C09099=1090.763,165.614,-68.521,176.010,19.399,152.921
C09100=1090.757,165.365,-68.500,176.007,19.398,152.921
C09101=1090.752,165.116,-68.478,176.005,19.397,152.921
C09102=1090.746,164.867,-68.456,176.002,19.396,152.921
C09103=1090.741,164.618,-68.434,175.999,19.395,152.922
C09104=1090.735,164.369,-68.413,175.996,19.394,152.922
C09105=1090.731,164.119,-68.391,175.994,19.392,152.922
C09106=1090.725,163.871,-68.370,175.991,19.391,152.922
C09107=1090.719,163.622,-68.348,175.988,19.390,152.923
C09108=1090.714,163.373,-68.327,175.986,19.389,152.923
C09109=1090.709,163.124,-68.305,175.983,19.388,152.923
C09110=1090.703,162.874,-68.284,175.981,19.387,152.923
C09111=1090.698,162.626,-68.263,175.978,19.386,152.923
C09112=1090.692,162.377,-68.241,175.976,19.385,152.924
C09113=1090.687,162.128,-68.219,175.973,19.383,152.924
C09114=1090.681,161.879,-68.198,175.970,19.382,152.924
C09115=1090.676,161.629,-68.176,175.967,19.381,152.924
C09116=1090.671,161.381,-68.155,175.965,19.380,152.925
C09117=1090.665,161.132,-68.134,175.962,19.379,152.925
C09118=1090.659,160.882,-68.113,175.959,19.378,152.925
C09119=1090.654,160.634,-68.092,175.957,19.377,152.925
C09120=1090.647,160.385,-68.070,175.955,19.376,152.926
C09121=1090.642,160.108,-68.046,175.952,19.375,152.926
C09122=1090.635,159.831,-68.023,175.948,19.373,152.926
C09123=1090.629,159.553,-67.999,175.946,19.372,152.926
C09124=1090.623,159.277,-67.975,175.943,19.371,152.927
C09125=1090.617,159.028,-67.954,175.940,19.370,152.927
C09126=1090.612,158.778,-67.933,175.937,19.369,152.927
C09127=1090.606,158.530,-67.912,175.935,19.368,152.927
C09128=1090.600,158.280,-67.891,175.932,19.367,152.927
C09129=1090.595,158.031,-67.870,175.930,19.366,152.928
C09130=1090.590,157.783,-67.848,175.927,19.365,152.928
C09131=1090.584,157.533,-67.827,175.925,19.364,152.928
C09132=1090.578,157.284,-67.806,175.922,19.362,152.928
C09133=1090.573,157.035,-67.785,175.919,19.361,152.929
C09134=1090.567,156.786,-67.763,175.916,19.360,152.929
C09135=1090.562,156.537,-67.743,175.914,19.359,152.929
C09136=1090.556,156.288,-67.722,175.912,19.358,152.929
C09137=1090.550,156.039,-67.700,175.909,19.357,152.929
C09138=1090.545,155.790,-67.679,175.906,19.356,152.930
C09139=1090.539,155.541,-67.658,175.904,19.355,152.930
C09140=1090.533,155.292,-67.637,175.901,19.353,152.930
C09141=1090.528,155.043,-67.616,175.898,19.352,152.930
C09142=1090.522,154.794,-67.595,175.896,19.351,152.931
C09143=1090.517,154.544,-67.574,175.894,19.351,152.931
C09144=1090.511,154.296,-67.553,175.891,19.349,152.931
C09145=1090.506,154.047,-67.533,175.888,19.348,152.931
C09146=1090.500,153.797,-67.511,175.886,19.347,152.932
C09147=1090.494,153.548,-67.490,175.883,19.346,152.932
C09148=1090.489,153.300,-67.469,175.880,19.344,152.932
C09149=1090.483,153.051,-67.449,175.878,19.344,152.932
C09150=1090.478,152.801,-67.428,175.876,19.343,152.932
C09151=1090.472,152.552,-67.406,175.873,19.341,152.933
C09152=1090.467,152.303,-67.386,175.870,19.340,152.933
C09153=1090.461,152.053,-67.365,175.868,19.339,152.933
C09154=1090.455,151.805,-67.344,175.865,19.338,152.933
C09155=1090.449,151.556,-67.324,175.863,19.337,152.933
C09156=1090.444,151.307,-67.303,175.860,19.336,152.934
C09157=1090.438,151.058,-67.282,175.858,19.334,152.934
C09158=1090.433,150.809,-67.261,175.855,19.333,152.934
C09159=1090.427,150.559,-67.240,175.852,19.332,152.934
C09160=1090.422,150.311,-67.219,175.850,19.331,152.934
C09161=1090.416,150.061,-67.198,175.848,19.330,152.935
C09162=1090.411,149.812,-67.178,175.845,19.329,152.935
C09163=1090.404,149.564,-67.157,175.843,19.328,152.935
C09164=1090.399,149.315,-67.136,175.840,19.327,152.935
C09165=1090.394,149.066,-67.116,175.837,19.325,152.936
C09166=1090.388,148.816,-67.095,175.835,19.324,152.936
C09167=1090.383,148.567,-67.074,175.833,19.323,152.936
C09168=1090.377,148.318,-67.053,175.830,19.322,152.936
C09169=1090.371,148.069,-67.033,175.827,19.321,152.936
C09170=1090.366,147.820,-67.013,175.825,19.320,152.937
C09171=1090.360,147.570,-66.992,175.822,19.318,152.937
C09172=1090.355,147.321,-66.971,175.820,19.318,152.937
C09173=1090.349,147.073,-66.951,175.817,19.317,152.937
C09174=1090.343,146.824,-66.930,175.815,19.315,152.937
C09175=1090.338,146.574,-66.909,175.812,19.314,152.938
C09176=1090.332,146.325,-66.889,175.809,19.312,152.938
C09177=1090.326,146.076,-66.869,175.808,19.312,152.938
C09178=1090.321,145.827,-66.848,175.805,19.311,152.938
C09179=1090.316,145.578,-66.827,175.802,19.309,152.938
C09180=1090.310,145.329,-66.807,175.799,19.308,152.939
C09181=1090.304,145.079,-66.787,175.797,19.307,152.939
C09182=1090.298,144.831,-66.765,175.795,19.306,152.939
C09183=1090.292,144.582,-66.745,175.792,19.305,152.939
C09184=1090.287,144.333,-66.725,175.790,19.303,152.939
C09185=1090.280,144.055,-66.702,175.787,19.302,152.940
C09186=1090.275,143.778,-66.679,175.784,19.301,152.940
C09187=1090.268,143.501,-66.657,175.782,19.300,152.940
C09188=1090.262,143.223,-66.634,175.779,19.298,152.940
C09189=1090.256,142.974,-66.614,175.776,19.297,152.940
C09190=1090.251,142.725,-66.594,175.774,19.296,152.940
C09191=1090.246,142.476,-66.573,175.771,19.295,152.941
C09192=1090.240,142.227,-66.553,175.769,19.293,152.941
C09193=1090.235,141.978,-66.533,175.767,19.292,152.941
C09194=1090.229,141.729,-66.512,175.764,19.291,152.941
C09195=1090.223,141.480,-66.492,175.761,19.290,152.941
C09196=1090.217,141.230,-66.471,175.759,19.288,152.942
C09197=1090.212,140.981,-66.451,175.757,19.288,152.942
C09198=1090.206,140.732,-66.431,175.754,19.286,152.942
C09199=1090.201,140.483,-66.410,175.752,19.285,152.942
C09200=1090.195,140.234,-66.390,175.749,19.284,152.942
C09201=1090.190,139.985,-66.370,175.746,19.283,152.943
C09202=1090.184,139.736,-66.350,175.745,19.282,152.943
C09203=1090.179,139.487,-66.330,175.742,19.280,152.943
C09204=1090.173,139.238,-66.310,175.739,19.279,152.943
C09205=1090.168,138.989,-66.289,175.737,19.277,152.943
C09206=1090.162,138.740,-66.269,175.735,19.277,152.943
C09207=1090.156,138.491,-66.249,175.732,19.275,152.944
C09208=1090.151,138.241,-66.230,175.730,19.274,152.944
C09209=1090.145,137.992,-66.209,175.727,19.273,152.944
C09210=1090.139,137.743,-66.189,175.725,19.272,152.944
C09211=1090.133,137.494,-66.168,175.723,19.271,152.944
C09212=1090.127,137.245,-66.148,175.720,19.270,152.945
C09213=1090.123,136.995,-66.128,175.717,19.268,152.945
C09214=1090.117,136.746,-66.108,175.715,19.266,152.945
C09215=1090.111,136.497,-66.088,175.713,19.266,152.945
C09216=1090.105,136.248,-66.068,175.710,19.264,152.945
C09217=1090.100,135.999,-66.049,175.708,19.263,152.945
C09218=1090.094,135.750,-66.028,175.705,19.262,152.946
C09219=1090.088,135.501,-66.008,175.703,19.261,152.946
C09220=1090.083,135.251,-65.988,175.701,19.260,152.946
C09221=1090.077,135.002,-65.968,175.698,19.258,152.946
C09222=1090.071,134.753,-65.948,175.695,19.257,152.946
C09223=1090.066,134.504,-65.928,175.694,19.256,152.946
C09224=1090.060,134.255,-65.909,175.691,19.254,152.946
C09225=1090.054,134.006,-65.889,175.688,19.253,152.947
C09226=1090.050,133.756,-65.869,175.686,19.252,152.947
C09227=1090.044,133.508,-65.849,175.684,19.251,152.947
C09228=1090.038,133.258,-65.828,175.681,19.250,152.947
C09229=1090.033,133.009,-65.809,175.679,19.248,152.947
C09230=1090.027,132.760,-65.789,175.676,19.247,152.947
C09231=1090.022,132.510,-65.769,175.674,19.246,152.948
C09232=1090.016,132.262,-65.749,175.672,19.245,152.948
C09233=1090.010,132.012,-65.730,175.669,19.243,152.948
C09234=1090.005,131.763,-65.709,175.667,19.242,152.948
C09235=1089.999,131.514,-65.689,175.665,19.241,152.948
C09236=1089.993,131.265,-65.670,175.662,19.239,152.948
C09237=1089.987,131.016,-65.650,175.660,19.238,152.949
C09238=1089.981,130.767,-65.631,175.658,19.237,152.949
C09239=1089.975,130.518,-65.611,175.655,19.236,152.949
C09240=1089.970,130.268,-65.591,175.653,19.235,152.949
C09241=1089.965,130.020,-65.572,175.650,19.233,152.949
C09242=1089.959,129.770,-65.552,175.648,19.233,152.950
C09243=1089.953,129.522,-65.532,175.646,19.231,152.950
C09244=1089.948,129.272,-65.513,175.643,19.229,152.950
C09245=1089.942,129.023,-65.493,175.641,19.229,152.950
C09246=1089.936,128.774,-65.474,175.639,19.227,152.950
C09247=1089.931,128.524,-65.454,175.636,19.226,152.950
C09248=1089.925,128.275,-65.434,175.634,19.224,152.950
C09249=1089.919,127.998,-65.413,175.631,19.223,152.951
C09250=1089.911,127.720,-65.391,175.628,19.222,152.951
C09251=1089.906,127.443,-65.369,175.626,19.220,152.951
C09252=1089.899,127.166,-65.347,175.623,19.219,152.951
C09253=1089.894,126.917,-65.328,175.621,19.218,152.951
C09254=1089.888,126.668,-65.308,175.619,19.217,152.951
C09255=1089.883,126.418,-65.288,175.616,19.215,152.952
C09256=1089.878,126.169,-65.269,175.613,19.214,152.952
C09257=1089.872,125.920,-65.249,175.612,19.213,152.952
C09258=1089.866,125.671,-65.230,175.609,19.211,152.952
C09259=1089.860,125.422,-65.211,175.607,19.210,152.952
C09260=1089.854,125.173,-65.191,175.605,19.209,152.952
C09261=1089.848,124.923,-65.172,175.602,19.208,152.952
C09262=1089.843,124.674,-65.152,175.600,19.206,152.953
C09263=1089.837,124.424,-65.133,175.598,19.205,152.953
C09264=1089.832,124.176,-65.114,175.596,19.204,152.953
C09265=1089.826,123.927,-65.094,175.593,19.202,152.953
C09266=1089.820,123.677,-65.075,175.590,19.201,152.953
C09267=1089.815,123.428,-65.056,175.589,19.200,152.953
C09268=1089.809,123.179,-65.036,175.586,19.198,152.953
C09269=1089.804,122.929,-65.016,175.584,19.197,152.954
C09270=1089.799,122.681,-64.997,175.582,19.196,152.954
C09271=1089.793,122.431,-64.978,175.579,19.194,152.954
C09272=1089.787,122.182,-64.959,175.577,19.193,152.954
C09273=1089.781,121.933,-64.939,175.575,19.192,152.954
C09274=1089.776,121.684,-64.919,175.572,19.191,152.954
C09275=1089.770,121.435,-64.901,175.570,19.189,152.954
C09276=1089.765,121.185,-64.881,175.567,19.188,152.954
C09277=1089.759,120.936,-64.862,175.566,19.186,152.955
C09278=1089.753,120.687,-64.843,175.563,19.185,152.955
C09279=1089.748,120.438,-64.824,175.561,19.183,152.955
C09280=1089.742,120.189,-64.804,175.559,19.182,152.955
C09281=1089.737,119.940,-64.785,175.556,19.181,152.955
C09282=1089.731,119.690,-64.766,175.554,19.179,152.955
C09283=1089.726,119.441,-64.747,175.552,19.178,152.955
C09284=1089.720,119.192,-64.727,175.550,19.177,152.955
C09285=1089.715,118.943,-64.708,175.547,19.176,152.956
C09286=1089.709,118.693,-64.689,175.545,19.175,152.956
C09287=1089.704,118.444,-64.670,175.543,19.173,152.956
C09288=1089.698,118.195,-64.651,175.540,19.171,152.956
C09289=1089.692,117.946,-64.632,175.538,19.170,152.956
C09290=1089.687,117.696,-64.612,175.536,19.169,152.956
C09291=1089.682,117.447,-64.593,175.533,19.167,152.956
C09292=1089.676,117.198,-64.574,175.532,19.166,152.956
C09293=1089.669,116.949,-64.556,175.529,19.165,152.957
C09294=1089.664,116.700,-64.537,175.527,19.163,152.957
C09295=1089.659,116.451,-64.517,175.525,19.162,152.957
C09296=1089.653,116.201,-64.498,175.523,19.160,152.957
C09297=1089.648,115.953,-64.479,175.520,19.159,152.957
C09298=1089.642,115.703,-64.460,175.518,19.158,152.957
C09299=1089.637,115.454,-64.441,175.516,19.156,152.957
C09300=1089.631,115.205,-64.422,175.513,19.154,152.957
C09301=1089.626,114.956,-64.403,175.512,19.153,152.957
C09302=1089.620,114.706,-64.383,175.509,19.152,152.957
C09303=1089.615,114.457,-64.365,175.507,19.150,152.958
C09304=1089.610,114.207,-64.346,175.505,19.149,152.958
C09305=1089.603,113.958,-64.327,175.503,19.148,152.958
C09306=1089.598,113.709,-64.308,175.500,19.146,152.958
C09307=1089.592,113.460,-64.289,175.498,19.145,152.958
C09308=1089.587,113.211,-64.270,175.496,19.144,152.958
C09309=1089.581,112.962,-64.252,175.493,19.142,152.958
C09310=1089.575,112.713,-64.232,175.492,19.141,152.958
C09311=1089.570,112.463,-64.214,175.489,19.139,152.958
C09312=1089.565,112.214,-64.195,175.487,19.138,152.959
C09313=1089.558,111.937,-64.174,175.484,19.136,152.959
C09314=1089.551,111.659,-64.153,175.481,19.135,152.959
C09315=1089.545,111.382,-64.132,175.479,19.133,152.959
C09316=1089.539,111.104,-64.112,175.477,19.131,152.959
C09317=1089.534,110.855,-64.093,175.475,19.130,152.959
C09318=1089.527,110.606,-64.074,175.472,19.129,152.959
C09319=1089.522,110.357,-64.055,175.471,19.128,152.959
C09320=1089.517,110.107,-64.037,175.468,19.126,152.959
C09321=1089.511,109.858,-64.018,175.466,19.125,152.960
C09322=1089.505,109.609,-63.999,175.464,19.123,152.960
C09323=1089.499,109.360,-63.981,175.462,19.122,152.960
C09324=1089.494,109.110,-63.962,175.459,19.120,152.960
C09325=1089.488,108.861,-63.943,175.457,19.119,152.960
C09326=1089.482,108.612,-63.925,175.455,19.118,152.960
C09327=1089.477,108.362,-63.906,175.452,19.116,152.960
C09328=1089.471,108.114,-63.888,175.451,19.115,152.960
C09329=1089.465,107.865,-63.869,175.448,19.114,152.960
C09330=1089.460,107.614,-63.850,175.447,19.112,152.960
C09331=1089.454,107.366,-63.832,175.444,19.111,152.961
C09332=1089.448,107.117,-63.813,175.442,19.109,152.961
C09333=1089.443,106.868,-63.795,175.440,19.108,152.961
C09334=1089.437,106.618,-63.776,175.437,19.106,152.961
C09335=1089.431,106.368,-63.758,175.435,19.105,152.961
C09336=1089.426,106.120,-63.739,175.433,19.104,152.961
C09337=1089.420,105.870,-63.720,175.431,19.102,152.961
C09338=1089.415,105.621,-63.702,175.429,19.101,152.961
C09339=1089.409,105.372,-63.683,175.427,19.099,152.961
C09340=1089.404,105.123,-63.665,175.424,19.098,152.961
C09341=1089.398,104.873,-63.646,175.422,19.097,152.962
C09342=1089.392,104.624,-63.628,175.420,19.095,152.961
C09343=1089.387,104.375,-63.609,175.418,19.093,152.962
C09344=1089.381,104.125,-63.591,175.416,19.092,152.962
C09345=1089.375,103.876,-63.572,175.413,19.090,152.962
C09346=1089.369,103.627,-63.554,175.412,19.089,152.962
C09347=1089.364,103.378,-63.536,175.410,19.087,152.962
C09348=1089.358,103.128,-63.518,175.407,19.086,152.962
C09349=1089.353,102.879,-63.499,175.405,19.085,152.962
C09350=1089.347,102.630,-63.481,175.403,19.083,152.962
C09351=1089.342,102.381,-63.462,175.401,19.081,152.962
C09352=1089.336,102.131,-63.443,175.399,19.080,152.962
C09353=1089.331,101.882,-63.425,175.396,19.079,152.962
C09354=1089.325,101.633,-63.407,175.395,19.078,152.963
C09355=1089.320,101.383,-63.389,175.392,19.076,152.963
C09356=1089.313,101.134,-63.370,175.390,19.074,152.963
C09357=1089.309,100.885,-63.352,175.388,19.073,152.963
C09358=1089.302,100.636,-63.334,175.386,19.071,152.963
C09359=1089.297,100.387,-63.316,175.384,19.070,152.963
C09360=1089.291,100.137,-63.298,175.382,19.068,152.963
C09361=1089.285,99.888,-63.279,175.379,19.067,152.963
C09362=1089.279,99.639,-63.261,175.377,19.066,152.963
C09363=1089.274,99.390,-63.242,175.375,19.064,152.963
C09364=1089.268,99.140,-63.225,175.374,19.063,152.963
C09365=1089.263,98.891,-63.207,175.371,19.061,152.963
C09366=1089.257,98.641,-63.188,175.368,19.060,152.964
C09367=1089.251,98.393,-63.170,175.367,19.058,152.963
C09368=1089.245,98.143,-63.152,175.365,19.057,152.964
C09369=1089.240,97.893,-63.134,175.363,19.055,152.964
C09370=1089.235,97.645,-63.116,175.360,19.054,152.964
C09371=1089.228,97.395,-63.098,175.358,19.052,152.964
C09372=1089.223,97.146,-63.080,175.356,19.051,152.964
C09373=1089.218,96.896,-63.062,175.354,19.049,152.964
C09374=1089.212,96.648,-63.043,175.352,19.048,152.964
C09375=1089.206,96.398,-63.026,175.350,19.046,152.964
C09376=1089.201,96.149,-63.007,175.347,19.045,152.964
C09377=1089.194,95.871,-62.988,175.346,19.043,152.964
C09378=1089.188,95.595,-62.967,175.343,19.042,152.964
C09379=1089.181,95.317,-62.947,175.341,19.040,152.964
C09380=1089.175,95.039,-62.927,175.339,19.038,152.964
C09381=1089.169,94.790,-62.909,175.336,19.036,152.965
C09382=1089.164,94.541,-62.891,175.335,19.035,152.965
C09383=1089.159,94.292,-62.873,175.332,19.033,152.965
C09384=1089.153,94.042,-62.855,175.330,19.032,152.965
C09385=1089.147,93.793,-62.838,175.328,19.030,152.965
C09386=1089.142,93.544,-62.820,175.326,19.029,152.965
C09387=1089.136,93.294,-62.801,175.324,19.027,152.965
C09388=1089.131,93.045,-62.784,175.322,19.026,152.965
C09389=1089.125,92.795,-62.766,175.320,19.025,152.965
C09390=1089.119,92.547,-62.748,175.318,19.023,152.965
C09391=1089.113,92.298,-62.730,175.316,19.022,152.965
C09392=1089.108,92.048,-62.712,175.314,19.019,152.965
C09393=1089.102,91.799,-62.694,175.311,19.018,152.965
C09394=1089.097,91.550,-62.676,175.310,19.016,152.965
C09395=1089.091,91.300,-62.658,175.307,19.015,152.965
C09396=1089.085,91.051,-62.641,175.306,19.014,152.965
C09397=1089.080,90.802,-62.623,175.303,19.012,152.965
C09398=1089.074,90.552,-62.605,175.302,19.011,152.965
C09399=1089.069,90.303,-62.587,175.299,19.009,152.965
C09400=1089.063,90.054,-62.570,175.297,19.007,152.966
C09401=1089.057,89.804,-62.552,175.295,19.006,152.966
C09402=1089.052,89.555,-62.534,175.293,19.004,152.966
C09403=1089.045,89.305,-62.516,175.291,19.003,152.966
C09404=1089.040,89.056,-62.499,175.289,19.001,152.966
C09405=1089.034,88.807,-62.481,175.287,19.000,152.966
C09406=1089.028,88.557,-62.463,175.285,18.998,152.966
C09407=1089.023,88.308,-62.446,175.282,18.996,152.966
C09408=1089.017,88.059,-62.428,175.281,18.995,152.966
C09409=1089.011,87.810,-62.410,175.279,18.993,152.966
C09410=1089.006,87.561,-62.393,175.277,18.992,152.966
C09411=1089.000,87.312,-62.375,175.275,18.990,152.966
C09412=1088.994,87.062,-62.357,175.273,18.989,152.966
C09413=1088.989,86.812,-62.340,175.271,18.987,152.966
C09414=1088.983,86.563,-62.323,175.269,18.986,152.966
C09415=1088.977,86.313,-62.305,175.266,18.984,152.966
C09416=1088.972,86.064,-62.287,175.264,18.982,152.966
C09417=1088.966,85.815,-62.270,175.262,18.981,152.967
C09418=1088.961,85.566,-62.252,175.260,18.979,152.967
C09419=1088.954,85.316,-62.234,175.259,18.978,152.967
C09420=1088.949,85.067,-62.217,175.256,18.976,152.967
C09421=1088.943,84.818,-62.200,175.255,18.975,152.967
C09422=1088.937,84.569,-62.183,175.252,18.973,152.967
C09423=1088.931,84.319,-62.165,175.251,18.972,152.967
C09424=1088.926,84.070,-62.147,175.248,18.970,152.967
C09425=1088.920,83.821,-62.130,175.247,18.969,152.967
C09426=1088.915,83.572,-62.113,175.244,18.967,152.967
C09427=1088.909,83.322,-62.095,175.242,18.965,152.967
C09428=1088.903,83.073,-62.077,175.240,18.964,152.967
C09429=1088.898,82.824,-62.060,175.238,18.962,152.967
C09430=1088.893,82.574,-62.043,175.236,18.961,152.967
C09431=1088.887,82.324,-62.025,175.234,18.959,152.967
C09432=1088.881,82.075,-62.007,175.233,18.957,152.967
C09433=1088.876,81.826,-61.990,175.230,18.956,152.967
C09434=1088.870,81.577,-61.973,175.229,18.954,152.967
C09435=1088.864,81.328,-61.956,175.226,18.953,152.967
C09436=1088.858,81.078,-61.938,175.225,18.951,152.967
C09437=1088.853,80.828,-61.921,175.223,18.949,152.967
C09438=1088.847,80.579,-61.904,175.221,18.948,152.967
C09439=1088.842,80.330,-61.886,175.219,18.946,152.967
C09440=1088.837,80.081,-61.869,175.216,18.944,152.967
C09441=1088.830,79.804,-61.850,175.215,18.943,152.967
C09442=1088.824,79.526,-61.830,175.212,18.941,152.967
C09443=1088.817,79.248,-61.811,175.210,18.939,152.967
C09444=1088.811,78.972,-61.792,175.208,18.937,152.967
C09445=1088.805,78.723,-61.775,175.206,18.936,152.967
C09446=1088.800,78.473,-61.758,175.204,18.934,152.967
C09447=1088.795,78.224,-61.740,175.202,18.933,152.967
C09448=1088.788,77.974,-61.724,175.200,18.931,152.967
C09449=1088.783,77.725,-61.706,175.198,18.929,152.967
C09450=1088.777,77.476,-61.689,175.196,18.927,152.967
C09451=1088.772,77.226,-61.672,175.195,18.926,152.967
C09452=1088.766,76.977,-61.655,175.192,18.924,152.968
C09453=1088.760,76.727,-61.637,175.191,18.923,152.968
C09454=1088.754,76.478,-61.620,175.188,18.921,152.968
C09455=1088.748,76.229,-61.604,175.187,18.920,152.968
C09456=1088.743,75.980,-61.586,175.184,18.918,152.968
C09457=1088.738,75.730,-61.569,175.182,18.916,152.968
C09458=1088.731,75.481,-61.552,175.180,18.915,152.968
C09459=1088.726,75.232,-61.535,175.178,18.913,152.968
C09460=1088.720,74.982,-61.517,175.177,18.911,152.968
C09461=1088.714,74.732,-61.501,175.174,18.909,152.968
C09462=1088.708,74.483,-61.484,175.173,18.908,152.968
C09463=1088.703,74.234,-61.467,175.170,18.906,152.968
C09464=1088.697,73.985,-61.450,175.169,18.905,152.968
C09465=1088.692,73.735,-61.433,175.167,18.903,152.968
C09466=1088.686,73.486,-61.415,175.165,18.902,152.968
C09467=1088.680,73.237,-61.399,175.163,18.900,152.968
C09468=1088.675,72.987,-61.382,175.161,18.898,152.968
C09469=1088.669,72.738,-61.364,175.159,18.897,152.968
C09470=1088.663,72.488,-61.348,175.157,18.895,152.968
C09471=1088.658,72.239,-61.331,175.155,18.893,152.968
C09472=1088.652,71.989,-61.314,175.153,18.892,152.968
C09473=1088.646,71.740,-61.297,175.151,18.890,152.968
C09474=1088.641,71.491,-61.280,175.150,18.888,152.968
C09475=1088.635,71.242,-61.264,175.147,18.886,152.968
C09476=1088.630,70.992,-61.247,175.146,18.885,152.968
C09477=1088.624,70.743,-61.229,175.143,18.883,152.968
C09478=1088.618,70.494,-61.213,175.142,18.882,152.968
C09479=1088.613,70.244,-61.196,175.140,18.880,152.968
C09480=1088.607,69.995,-61.179,175.138,18.879,152.968
C09481=1088.602,69.746,-61.162,175.136,18.877,152.968
C09482=1088.595,69.496,-61.146,175.134,18.875,152.968
C09483=1088.589,69.247,-61.128,175.132,18.873,152.968
C09484=1088.584,68.997,-61.112,175.130,18.872,152.968
C09485=1088.578,68.748,-61.095,175.128,18.870,152.968
C09486=1088.572,68.498,-61.079,175.127,18.868,152.968
C09487=1088.567,68.249,-61.061,175.124,18.867,152.968
C09488=1088.561,68.000,-61.045,175.123,18.865,152.968
C09489=1088.556,67.750,-61.028,175.120,18.863,152.968
C09490=1088.550,67.501,-61.012,175.119,18.862,152.968
C09491=1088.544,67.252,-60.994,175.117,18.860,152.968
C09492=1088.538,67.002,-60.978,175.115,18.859,152.968
C09493=1088.533,66.753,-60.961,175.113,18.856,152.968
C09494=1088.527,66.503,-60.945,175.111,18.855,152.968
C09495=1088.521,66.254,-60.929,175.110,18.853,152.968
C09496=1088.516,66.005,-60.911,175.107,18.852,152.968
C09497=1088.510,65.756,-60.895,175.106,18.850,152.968
C09498=1088.504,65.506,-60.878,175.104,18.848,152.968
C09499=1088.499,65.257,-60.862,175.102,18.847,152.968
C09500=1088.493,65.007,-60.845,175.100,18.845,152.968
C09501=1088.487,64.758,-60.829,175.098,18.844,152.968
C09502=1088.481,64.509,-60.812,175.096,18.842,152.968
C09503=1088.476,64.259,-60.795,175.095,18.840,152.968
C09504=1088.470,64.010,-60.778,175.092,18.838,152.968
C09505=1088.464,63.732,-60.760,175.090,18.836,152.968
C09506=1088.457,63.455,-60.742,175.088,18.835,152.968
C09507=1088.451,63.178,-60.724,175.086,18.833,152.968
C09508=1088.444,62.900,-60.705,175.084,18.831,152.968
C09509=1088.438,62.651,-60.689,175.083,18.829,152.968
C09510=1088.432,62.402,-60.673,175.080,18.828,152.968
C09511=1088.426,62.152,-60.656,175.079,18.826,152.968
C09512=1088.421,61.903,-60.640,175.076,18.824,152.968
C09513=1088.415,61.653,-60.623,175.075,18.823,152.968
C09514=1088.409,61.404,-60.607,175.072,18.821,152.968
C09515=1088.403,61.155,-60.591,175.071,18.819,152.968
C09516=1088.397,60.905,-60.575,175.069,18.818,152.968
C09517=1088.392,60.656,-60.558,175.067,18.816,152.968
C09518=1088.386,60.406,-60.541,175.066,18.814,152.968
C09519=1088.380,60.157,-60.525,175.063,18.813,152.968
C09520=1088.374,59.907,-60.509,175.062,18.811,152.968
C09521=1088.368,59.658,-60.493,175.060,18.809,152.968
C09522=1088.363,59.408,-60.476,175.058,18.808,152.968
C09523=1088.357,59.159,-60.460,175.056,18.806,152.968
C09524=1088.351,58.910,-60.443,175.054,18.804,152.968
C09525=1088.345,58.660,-60.427,175.052,18.802,152.968
C09526=1088.339,58.411,-60.411,175.051,18.801,152.968
C09527=1088.333,58.162,-60.395,175.048,18.799,152.968
C09528=1088.328,57.912,-60.378,175.047,18.797,152.968
C09529=1088.322,57.663,-60.361,175.045,18.796,152.968
C09530=1088.316,57.413,-60.345,175.043,18.794,152.968
C09531=1088.311,57.165,-60.329,175.041,18.793,152.968
C09532=1088.305,56.915,-60.314,175.039,18.791,152.968
C09533=1088.299,56.665,-60.298,175.038,18.789,152.968
C09534=1088.294,56.416,-60.281,175.035,18.787,152.968
C09535=1088.288,56.166,-60.264,175.034,18.786,152.968
C09536=1088.282,55.917,-60.248,175.032,18.783,152.968
C09537=1088.276,55.668,-60.232,175.030,18.782,152.968
C09538=1088.270,55.418,-60.216,175.029,18.780,152.968
C09539=1088.265,55.168,-60.200,175.027,18.778,152.968
C09540=1088.259,54.920,-60.184,175.025,18.777,152.968
C09541=1088.253,54.670,-60.168,175.023,18.775,152.968
C09542=1088.248,54.421,-60.151,175.021,18.774,152.968
C09543=1088.242,54.171,-60.135,175.019,18.772,152.968
C09544=1088.237,53.921,-60.119,175.018,18.770,152.968
C09545=1088.231,53.672,-60.103,175.015,18.768,152.968
C09546=1088.225,53.423,-60.087,175.014,18.766,152.968
C09547=1088.219,53.174,-60.071,175.013,18.765,152.968
C09548=1088.214,52.924,-60.055,175.010,18.763,152.968
C09549=1088.208,52.675,-60.039,175.009,18.761,152.968
C09550=1088.202,52.425,-60.023,175.007,18.759,152.968
C09551=1088.196,52.175,-60.007,175.005,18.758,152.968
C09552=1088.191,51.927,-59.991,175.003,18.756,152.968
C09553=1088.186,51.677,-59.975,175.001,18.754,152.968
C09554=1088.180,51.428,-59.958,175.000,18.753,152.968
C09555=1088.174,51.178,-59.943,174.998,18.751,152.968
C09556=1088.168,50.928,-59.927,174.996,18.749,152.967
C09557=1088.163,50.680,-59.911,174.994,18.747,152.967
C09558=1088.157,50.430,-59.895,174.993,18.745,152.967
C09559=1088.151,50.181,-59.879,174.990,18.743,152.967
C09560=1088.145,49.931,-59.863,174.989,18.742,152.967
C09561=1088.140,49.681,-59.847,174.987,18.740,152.967
C09562=1088.134,49.433,-59.831,174.985,18.738,152.967
C09563=1088.129,49.183,-59.816,174.984,18.737,152.967
C09564=1088.123,48.933,-59.799,174.982,18.735,152.967
C09565=1088.117,48.684,-59.783,174.980,18.733,152.967
C09566=1088.112,48.435,-59.768,174.978,18.731,152.967
C09567=1088.106,48.185,-59.752,174.976,18.729,152.967
C09568=1088.100,47.935,-59.736,174.974,18.727,152.967
C09569=1088.094,47.658,-59.718,174.973,18.726,152.967
C09570=1088.088,47.381,-59.701,174.971,18.724,152.967
C09571=1088.082,47.103,-59.683,174.968,18.722,152.967
C09572=1088.075,46.825,-59.665,174.967,18.720,152.967
C09573=1088.069,46.575,-59.650,174.965,18.718,152.967
C09574=1088.064,46.327,-59.634,174.963,18.716,152.967
C09575=1088.058,46.077,-59.618,174.961,18.714,152.967
C09576=1088.052,45.827,-59.602,174.960,18.712,152.967
C09577=1088.047,45.578,-59.587,174.958,18.711,152.967
C09578=1088.041,45.329,-59.571,174.956,18.709,152.967
C09579=1088.036,45.079,-59.555,174.955,18.707,152.967
C09580=1088.030,44.830,-59.539,174.952,18.705,152.967
C09581=1088.025,44.580,-59.524,174.951,18.704,152.967
C09582=1088.019,44.331,-59.507,174.949,18.702,152.967
C09583=1088.014,44.082,-59.492,174.947,18.700,152.967
C09584=1088.008,43.832,-59.476,174.946,18.699,152.967
C09585=1088.002,43.582,-59.460,174.944,18.696,152.967
C09586=1087.997,43.333,-59.445,174.942,18.694,152.966
C09587=1087.991,43.084,-59.429,174.940,18.692,152.966
C09588=1087.985,42.834,-59.414,174.939,18.691,152.966
C09589=1087.979,42.585,-59.398,174.937,18.689,152.966
C09590=1087.974,42.335,-59.383,174.935,18.687,152.966
C09591=1087.968,42.085,-59.367,174.934,18.686,152.966
C09592=1087.962,41.836,-59.351,174.931,18.684,152.966
C09593=1087.956,41.587,-59.336,174.930,18.682,152.966
C09594=1087.950,41.338,-59.320,174.928,18.681,152.966
C09595=1087.945,41.088,-59.304,174.926,18.678,152.966
C09596=1087.940,40.839,-59.289,174.925,18.677,152.966
C09597=1087.934,40.589,-59.273,174.923,18.675,152.966
C09598=1087.927,40.340,-59.258,174.921,18.673,152.966
C09599=1087.922,40.090,-59.243,174.920,18.672,152.966
C09600=1087.916,39.841,-59.227,174.917,18.670,152.966
C09601=1087.911,39.591,-59.211,174.916,18.668,152.966
C09602=1087.905,39.342,-59.196,174.914,18.666,152.966
C09603=1087.899,39.093,-59.180,174.913,18.664,152.966
C09604=1087.893,38.843,-59.165,174.911,18.662,152.966
C09605=1087.888,38.593,-59.150,174.909,18.660,152.966
C09606=1087.882,38.344,-59.135,174.907,18.659,152.966
C09607=1087.877,38.095,-59.119,174.906,18.657,152.966
C09608=1087.871,37.845,-59.103,174.904,18.655,152.966
C09609=1087.864,37.596,-59.088,174.902,18.654,152.965
C09610=1087.859,37.346,-59.073,174.900,18.652,152.965
C09611=1087.853,37.097,-59.057,174.899,18.650,152.965
C09612=1087.847,36.847,-59.042,174.897,18.649,152.965
C09613=1087.842,36.598,-59.027,174.895,18.646,152.965
C09614=1087.836,36.348,-59.011,174.894,18.645,152.965
C09615=1087.830,36.098,-58.996,174.891,18.643,152.965
C09616=1087.825,35.850,-58.980,174.890,18.641,152.965
C09617=1087.818,35.600,-58.965,174.889,18.639,152.965
C09618=1087.813,35.351,-58.950,174.886,18.637,152.965
C09619=1087.807,35.101,-58.935,174.885,18.636,152.965
C09620=1087.801,34.851,-58.920,174.884,18.634,152.965
C09621=1087.796,34.602,-58.904,174.881,18.632,152.965
C09622=1087.789,34.353,-58.889,174.880,18.631,152.965
C09623=1087.784,34.104,-58.874,174.878,18.628,152.965
C09624=1087.778,33.854,-58.859,174.876,18.627,152.965
C09625=1087.772,33.604,-58.843,174.875,18.625,152.965
C09626=1087.767,33.355,-58.829,174.873,18.623,152.965
C09627=1087.761,33.105,-58.813,174.871,18.621,152.965
C09628=1087.756,32.856,-58.798,174.870,18.620,152.965
C09629=1087.750,32.606,-58.783,174.868,18.618,152.965
C09630=1087.745,32.357,-58.768,174.866,18.616,152.965
C09631=1087.738,32.107,-58.753,174.864,18.614,152.965
C09632=1087.732,31.858,-58.737,174.863,18.612,152.965
C09633=1087.726,31.580,-58.720,174.860,18.610,152.965
C09634=1087.720,31.302,-58.703,174.859,18.608,152.964
C09635=1087.714,31.025,-58.687,174.857,18.606,152.964
C09636=1087.706,30.748,-58.670,174.856,18.605,152.964
C09637=1087.701,30.499,-58.655,174.853,18.603,152.964
C09638=1087.696,30.249,-58.639,174.852,18.601,152.964
C09639=1087.690,30.000,-58.625,174.850,18.599,152.964
C09640=1087.684,29.750,-58.609,174.848,18.597,152.964
C09641=1087.678,29.501,-58.595,174.847,18.595,152.964
C09642=1087.673,29.251,-58.579,174.845,18.593,152.964
C09643=1087.667,29.002,-58.564,174.843,18.592,152.964
C09644=1087.661,28.752,-58.549,174.842,18.590,152.964
C09645=1087.656,28.503,-58.534,174.840,18.588,152.964
C09646=1087.649,28.253,-58.519,174.838,18.586,152.964
C09647=1087.644,28.004,-58.504,174.837,18.585,152.964
C09648=1087.638,27.754,-58.489,174.835,18.583,152.964
C09649=1087.633,27.504,-58.475,174.833,18.581,152.964
C09650=1087.627,27.255,-58.460,174.831,18.579,152.964
C09651=1087.621,27.006,-58.445,174.830,18.577,152.964
C09652=1087.615,26.756,-58.430,174.828,18.576,152.963
C09653=1087.609,26.506,-58.415,174.826,18.573,152.963
C09654=1087.603,26.257,-58.400,174.825,18.572,152.963
C09655=1087.597,26.007,-58.385,174.823,18.570,152.963
C09656=1087.592,25.758,-58.370,174.821,18.568,152.963
C09657=1087.585,25.509,-58.355,174.820,18.567,152.963
C09658=1087.581,25.259,-58.341,174.818,18.565,152.963
C09659=1087.575,25.010,-58.326,174.816,18.563,152.963
C09660=1087.568,24.760,-58.311,174.815,18.561,152.963
C09661=1087.563,24.511,-58.296,174.814,18.559,152.963
C09662=1087.557,24.261,-58.281,174.811,18.557,152.963
C09663=1087.551,24.012,-58.266,174.810,18.556,152.963
C09664=1087.546,23.762,-58.252,174.808,18.554,152.963
C09665=1087.540,23.513,-58.237,174.806,18.552,152.963
C09666=1087.534,23.263,-58.222,174.805,18.551,152.963
C09667=1087.529,23.014,-58.207,174.804,18.548,152.963
C09668=1087.522,22.764,-58.192,174.801,18.546,152.963
C09669=1087.517,22.514,-58.178,174.800,18.545,152.963
C09670=1087.510,22.265,-58.163,174.798,18.543,152.962
C09671=1087.505,22.016,-58.148,174.796,18.541,152.962
C09672=1087.500,21.767,-58.133,174.795,18.539,152.962
C09673=1087.493,21.516,-58.119,174.794,18.538,152.962
C09674=1087.488,21.267,-58.104,174.791,18.536,152.962
C09675=1087.482,21.017,-58.089,174.790,18.534,152.962
C09676=1087.477,20.768,-58.075,174.789,18.532,152.962
C09677=1087.471,20.519,-58.061,174.786,18.530,152.962
C09678=1087.465,20.269,-58.045,174.785,18.528,152.962
C09679=1087.459,20.020,-58.030,174.784,18.527,152.962
C09680=1087.453,19.770,-58.016,174.781,18.525,152.962
C09681=1087.448,19.521,-58.002,174.780,18.523,152.962
C09682=1087.441,19.271,-57.987,174.779,18.522,152.962
C09683=1087.436,19.021,-57.972,174.777,18.519,152.962
C09684=1087.431,18.772,-57.958,174.775,18.517,152.962
C09685=1087.424,18.523,-57.943,174.774,18.516,152.962
C09686=1087.419,18.273,-57.929,174.772,18.514,152.962
C09687=1087.412,18.023,-57.914,174.770,18.512,152.962
C09688=1087.407,17.774,-57.900,174.769,18.511,152.961
C09689=1087.401,17.525,-57.885,174.767,18.508,152.961
C09690=1087.395,17.275,-57.870,174.765,18.507,152.961
C09691=1087.390,17.025,-57.856,174.764,18.505,152.961
C09692=1087.384,16.776,-57.842,174.762,18.503,152.961
C09693=1087.378,16.526,-57.827,174.760,18.501,152.961
C09694=1087.372,16.277,-57.813,174.759,18.499,152.961
C09695=1087.366,16.027,-57.798,174.757,18.497,152.961
C09696=1087.360,15.778,-57.784,174.755,18.496,152.961
C09697=1087.354,15.502,-57.768,174.754,18.494,152.961
C09698=1087.348,15.226,-57.752,174.752,18.492,152.961
C09699=1087.341,14.949,-57.736,174.750,18.490,152.961
C09700=1087.335,14.674,-57.720,174.748,18.488,152.961
C09701=1087.330,14.424,-57.705,174.747,18.486,152.961
C09702=1087.324,14.175,-57.690,174.745,18.484,152.961
C09703=1087.317,13.925,-57.677,174.743,18.482,152.960
C09704=1087.312,13.676,-57.662,174.742,18.481,152.960
C09705=1087.306,13.425,-57.648,174.740,18.479,152.960
C09706=1087.300,13.177,-57.633,174.738,18.477,152.960
C09707=1087.294,12.927,-57.620,174.737,18.476,152.960
C09708=1087.288,12.677,-57.605,174.735,18.474,152.960
C09709=1087.282,12.428,-57.591,174.734,18.471,152.960
C09710=1087.277,12.178,-57.577,174.732,18.470,152.960
C09711=1087.271,11.928,-57.562,174.731,18.468,152.960
C09712=1087.265,11.679,-57.548,174.728,18.466,152.960
C09713=1087.259,11.430,-57.534,174.727,18.465,152.960
C09714=1087.253,11.180,-57.519,174.726,18.463,152.960
C09715=1087.248,10.931,-57.505,174.724,18.461,152.960
C09716=1087.242,10.681,-57.491,174.722,18.459,152.960
C09717=1087.236,10.431,-57.477,174.721,18.458,152.960
C09718=1087.230,10.182,-57.462,174.719,18.455,152.960
C09719=1087.224,9.933,-57.449,174.717,18.454,152.960
C09720=1087.218,9.683,-57.434,174.716,18.452,152.960
C09721=1087.212,9.433,-57.420,174.715,18.450,152.959
C09722=1087.207,9.184,-57.406,174.712,18.448,152.959
C09723=1087.200,8.934,-57.391,174.711,18.447,152.959
C09724=1087.195,8.685,-57.377,174.709,18.445,152.959
C09725=1087.189,8.435,-57.363,174.707,18.443,152.959
C09726=1087.183,8.185,-57.348,174.706,18.441,152.959
C09727=1087.177,7.936,-57.335,174.705,18.439,152.959
C09728=1087.171,7.687,-57.321,174.703,18.438,152.959
C09729=1087.165,7.438,-57.307,174.701,18.436,152.959
C09730=1087.159,7.187,-57.293,174.700,18.434,152.959
C09731=1087.154,6.938,-57.279,174.698,18.433,152.959
C09732=1087.148,6.688,-57.265,174.696,18.430,152.959
C09733=1087.143,6.439,-57.250,174.695,18.429,152.959
C09734=1087.137,6.189,-57.236,174.693,18.427,152.959
C09735=1087.131,5.939,-57.222,174.692,18.425,152.959
C09736=1087.125,5.690,-57.209,174.690,18.423,152.959
C09737=1087.119,5.441,-57.194,174.688,18.421,152.959
C09738=1087.113,5.191,-57.180,174.687,18.420,152.958
C09739=1087.108,4.941,-57.166,174.685,18.418,152.959
C09740=1087.102,4.692,-57.152,174.683,18.416,152.958
C09741=1087.096,4.443,-57.138,174.682,18.414,152.958
C09742=1087.090,4.193,-57.124,174.681,18.413,152.958
C09743=1087.084,3.943,-57.110,174.679,18.410,152.958
C09744=1087.079,3.694,-57.096,174.677,18.409,152.958
C09745=1087.073,3.444,-57.083,174.676,18.407,152.958
C09746=1087.068,3.194,-57.069,174.674,18.405,152.958
C09747=1087.062,2.946,-57.054,174.672,18.403,152.958
C09748=1087.055,2.696,-57.040,174.671,18.402,152.958
C09749=1087.049,2.446,-57.027,174.670,18.400,152.958
C09750=1087.044,2.196,-57.013,174.668,18.398,152.958
C09751=1087.039,1.947,-56.999,174.666,18.396,152.958
C09752=1087.033,1.697,-56.985,174.665,18.394,152.958
C09753=1087.027,1.448,-56.972,174.663,18.393,152.958
C09754=1087.020,1.198,-56.957,174.661,18.390,152.957
C09755=1087.015,0.949,-56.943,174.660,18.389,152.957
C09756=1087.009,0.699,-56.929,174.658,18.387,152.957
C09757=1087.004,0.450,-56.915,174.656,18.385,152.957
C09758=1086.998,0.200,-56.902,174.655,18.383,152.957
C09759=1086.992,-0.049,-56.888,174.654,18.381,152.957
C09760=1086.987,-0.299,-56.874,174.652,18.380,152.957
C09761=1086.980,-0.573,-56.859,174.650,18.378,152.957
C09762=1086.974,-0.847,-56.843,174.649,18.376,152.957
C09763=1086.968,-1.122,-56.829,174.647,18.374,152.957
C09764=1086.962,-1.396,-56.813,174.645,18.372,152.957
C09765=1086.956,-1.645,-56.800,174.643,18.370,152.957
C09766=1086.950,-1.894,-56.786,174.642,18.368,152.957
C09767=1086.944,-2.145,-56.772,174.640,18.366,152.957
C09768=1086.939,-2.394,-56.758,174.639,18.364,152.956
C09769=1086.932,-2.644,-56.745,174.637,18.362,152.956
C09770=1086.927,-2.893,-56.731,174.636,18.361,152.956
C09771=1086.921,-3.143,-56.717,174.634,18.359,152.956
C09772=1086.916,-3.392,-56.703,174.633,18.357,152.956
C09773=1086.910,-3.642,-56.690,174.631,18.355,152.956
C09774=1086.904,-3.891,-56.676,174.629,18.353,152.956
C09775=1086.898,-4.140,-56.663,174.628,18.352,152.956
C09776=1086.892,-4.391,-56.649,174.627,18.350,152.956
C09777=1086.886,-4.640,-56.635,174.624,18.348,152.956
C09778=1086.880,-4.890,-56.621,174.623,18.346,152.956
C09779=1086.874,-5.139,-56.608,174.622,18.345,152.956
C09780=1086.869,-5.388,-56.594,174.620,18.343,152.956
C09781=1086.862,-5.638,-56.581,174.618,18.341,152.956
C09782=1086.857,-5.888,-56.568,174.617,18.339,152.956
C09783=1086.851,-6.137,-56.555,174.615,18.338,152.956
C09784=1086.845,-6.387,-56.540,174.614,18.336,152.955
C09785=1086.839,-6.637,-56.527,174.612,18.334,152.955
C09786=1086.833,-6.886,-56.513,174.610,18.332,152.955
C09787=1086.827,-7.135,-56.500,174.609,18.331,152.955
C09788=1086.822,-7.385,-56.486,174.608,18.329,152.955
C09789=1086.815,-7.634,-56.473,174.605,18.327,152.955
C09790=1086.810,-7.885,-56.460,174.604,18.325,152.955
C09791=1086.804,-8.134,-56.446,174.603,18.323,152.955
C09792=1086.798,-8.383,-56.433,174.601,18.322,152.955
C09793=1086.792,-8.633,-56.419,174.599,18.320,152.955
C09794=1086.787,-8.882,-56.405,174.598,18.318,152.955
C09795=1086.780,-9.132,-56.392,174.597,18.316,152.955
C09796=1086.775,-9.382,-56.379,174.595,18.315,152.955
C09797=1086.769,-9.632,-56.365,174.593,18.313,152.955
C09798=1086.763,-9.881,-56.352,174.591,18.311,152.955
C09799=1086.757,-10.130,-56.338,174.590,18.309,152.955
C09800=1086.752,-10.381,-56.325,174.589,18.308,152.955
C09801=1086.745,-10.630,-56.312,174.588,18.306,152.954
C09802=1086.740,-10.879,-56.298,174.585,18.304,152.954
C09803=1086.734,-11.129,-56.285,174.584,18.302,152.954
C09804=1086.728,-11.379,-56.272,174.582,18.301,152.954
C09805=1086.722,-11.628,-56.258,174.581,18.299,152.954
C09806=1086.716,-11.877,-56.245,174.579,18.296,152.954
C09807=1086.711,-12.127,-56.231,174.578,18.295,152.954
C09808=1086.705,-12.377,-56.219,174.576,18.293,152.954
C09809=1086.699,-12.627,-56.205,174.575,18.292,152.954
C09810=1086.693,-12.876,-56.191,174.573,18.290,152.954
C09811=1086.688,-13.126,-56.178,174.571,18.288,152.954
C09812=1086.682,-13.375,-56.165,174.570,18.286,152.954
C09813=1086.676,-13.624,-56.152,174.569,18.284,152.954
C09814=1086.670,-13.875,-56.139,174.567,18.283,152.954
C09815=1086.664,-14.124,-56.125,174.565,18.281,152.954
C09816=1086.659,-14.374,-56.111,174.564,18.279,152.954
C09817=1086.653,-14.623,-56.099,174.562,18.277,152.954
C09818=1086.647,-14.873,-56.086,174.561,18.276,152.953
C09819=1086.641,-15.122,-56.072,174.559,18.274,152.953
C09820=1086.635,-15.372,-56.059,174.557,18.272,152.953
C09821=1086.629,-15.621,-56.046,174.556,18.270,152.953
C09822=1086.624,-15.872,-56.033,174.555,18.268,152.953
C09823=1086.618,-16.121,-56.020,174.553,18.267,152.953
C09824=1086.611,-16.370,-56.006,174.551,18.265,152.953
C09825=1086.605,-16.643,-55.992,174.550,18.263,152.953
C09826=1086.599,-16.915,-55.978,174.548,18.262,152.953
C09827=1086.592,-17.188,-55.964,174.546,18.259,152.953
C09828=1086.586,-17.460,-55.949,174.545,18.257,152.953
C09829=1086.580,-17.710,-55.937,174.543,18.256,152.953
C09830=1086.574,-17.959,-55.923,174.541,18.254,152.953
C09831=1086.568,-18.209,-55.910,174.540,18.252,152.953
C09832=1086.562,-18.458,-55.897,174.538,18.251,152.953
C09833=1086.556,-18.708,-55.884,174.537,18.249,152.953
C09834=1086.551,-18.958,-55.871,174.536,18.247,152.953
C09835=1086.545,-19.208,-55.858,174.534,18.245,152.953
C09836=1086.539,-19.457,-55.845,174.532,18.243,152.953
C09837=1086.533,-19.707,-55.832,174.531,18.242,152.952
C09838=1086.527,-19.956,-55.819,174.529,18.240,152.952
C09839=1086.522,-20.206,-55.806,174.528,18.239,152.952
C09840=1086.516,-20.455,-55.793,174.526,18.237,152.952
C09841=1086.510,-20.705,-55.780,174.525,18.235,152.952
C09842=1086.504,-20.954,-55.767,174.523,18.233,152.952
C09843=1086.498,-21.204,-55.754,174.522,18.232,152.952
C09844=1086.491,-21.453,-55.741,174.520,18.230,152.952
C09845=1086.486,-21.703,-55.728,174.518,18.228,152.952
C09846=1086.480,-21.953,-55.715,174.517,18.226,152.952
C09847=1086.474,-22.203,-55.702,174.515,18.225,152.952
C09848=1086.468,-22.452,-55.690,174.514,18.223,152.952
C09849=1086.463,-22.701,-55.677,174.513,18.221,152.952
C09850=1086.457,-22.951,-55.664,174.511,18.219,152.952
C09851=1086.452,-23.201,-55.651,174.509,18.217,152.952
C09852=1086.445,-23.450,-55.638,174.508,18.216,152.952
C09853=1086.439,-23.700,-55.625,174.506,18.214,152.952
C09854=1086.433,-23.950,-55.612,174.505,18.213,152.952
C09855=1086.427,-24.199,-55.599,174.503,18.211,152.952
C09856=1086.421,-24.449,-55.587,174.501,18.209,152.951
C09857=1086.416,-24.698,-55.573,174.500,18.207,152.951
C09858=1086.411,-24.948,-55.561,174.499,18.206,152.951
C09859=1086.405,-25.198,-55.548,174.497,18.204,152.951
C09860=1086.398,-25.447,-55.535,174.495,18.202,152.951
C09861=1086.393,-25.697,-55.522,174.494,18.200,152.951
C09862=1086.387,-25.947,-55.510,174.492,18.199,152.951
C09863=1086.381,-26.196,-55.497,174.491,18.197,152.951
C09864=1086.375,-26.445,-55.484,174.490,18.195,152.951
C09865=1086.370,-26.696,-55.471,174.488,18.194,152.951
C09866=1086.364,-26.945,-55.458,174.486,18.191,152.951
C09867=1086.358,-27.195,-55.445,174.485,18.190,152.951
C09868=1086.352,-27.445,-55.433,174.483,18.188,152.951
C09869=1086.346,-27.694,-55.421,174.482,18.187,152.951
C09870=1086.340,-27.943,-55.408,174.480,18.185,152.951
C09871=1086.334,-28.193,-55.395,174.479,18.184,152.951
C09872=1086.328,-28.443,-55.383,174.477,18.182,152.951
C09873=1086.322,-28.692,-55.370,174.475,18.180,152.951
C09874=1086.316,-28.942,-55.357,174.474,18.178,152.951
C09875=1086.310,-29.192,-55.345,174.473,18.177,152.951
C09876=1086.304,-29.441,-55.332,174.471,18.175,152.951
C09877=1086.299,-29.691,-55.320,174.470,18.174,152.951
C09878=1086.293,-29.941,-55.307,174.468,18.171,152.950
C09879=1086.286,-30.190,-55.294,174.466,18.170,152.950
C09880=1086.281,-30.440,-55.281,174.465,18.168,152.950
C09881=1086.275,-30.690,-55.269,174.463,18.166,152.950
C09882=1086.269,-30.939,-55.257,174.462,18.165,152.950
C09883=1086.263,-31.189,-55.244,174.461,18.163,152.950
C09884=1086.256,-31.438,-55.231,174.458,18.161,152.950
C09885=1086.251,-31.687,-55.219,174.457,18.160,152.950
C09886=1086.245,-31.937,-55.206,174.456,18.158,152.950
C09887=1086.239,-32.187,-55.194,174.454,18.157,152.950
C09888=1086.233,-32.436,-55.182,174.453,18.155,152.950
C09889=1086.227,-32.708,-55.168,174.451,18.153,152.950
C09890=1086.220,-32.980,-55.154,174.449,18.151,152.950
C09891=1086.214,-33.252,-55.140,174.448,18.150,152.950
C09892=1086.208,-33.523,-55.127,174.446,18.147,152.950
C09893=1086.202,-33.773,-55.114,174.444,18.146,152.950
C09894=1086.196,-34.022,-55.103,174.443,18.144,152.950
C09895=1086.190,-34.272,-55.090,174.442,18.143,152.950
C09896=1086.184,-34.522,-55.078,174.440,18.141,152.950
C09897=1086.178,-34.772,-55.065,174.439,18.139,152.950
C09898=1086.173,-35.021,-55.053,174.437,18.138,152.950
C09899=1086.167,-35.271,-55.040,174.435,18.136,152.950
C09900=1086.161,-35.520,-55.027,174.434,18.134,152.950
C09901=1086.154,-35.770,-55.015,174.432,18.133,152.950
C09902=1086.149,-36.019,-55.003,174.431,18.131,152.949
C09903=1086.143,-36.269,-54.990,174.430,18.130,152.949
C09904=1086.137,-36.519,-54.978,174.428,18.128,152.949
C09905=1086.131,-36.769,-54.965,174.427,18.126,152.949
C09906=1086.126,-37.018,-54.953,174.424,18.124,152.949
C09907=1086.120,-37.268,-54.940,174.423,18.123,152.949
C09908=1086.113,-37.517,-54.928,174.422,18.121,152.949
C09909=1086.108,-37.766,-54.916,174.420,18.120,152.949
C09910=1086.102,-38.016,-54.904,174.419,18.118,152.949
C09911=1086.096,-38.266,-54.891,174.417,18.116,152.949
C09912=1086.091,-38.516,-54.880,174.416,18.115,152.949
C09913=1086.085,-38.765,-54.868,174.414,18.113,152.949
C09914=1086.079,-39.015,-54.855,174.412,18.111,152.949
C09915=1086.073,-39.265,-54.843,174.411,18.110,152.949
C09916=1086.067,-39.514,-54.831,174.410,18.108,152.949
C09917=1086.061,-39.764,-54.818,174.408,18.107,152.949
C09918=1086.055,-40.014,-54.806,174.407,18.105,152.949
C09919=1086.049,-40.263,-54.794,174.405,18.103,152.949
C09920=1086.043,-40.513,-54.782,174.404,18.102,152.949
C09921=1086.037,-40.763,-54.769,174.402,18.100,152.949
C09922=1086.030,-41.012,-54.757,174.400,18.098,152.949
C09923=1086.025,-41.261,-54.745,174.399,18.097,152.949
C09924=1086.019,-41.511,-54.732,174.398,18.095,152.949
C09925=1086.013,-41.761,-54.721,174.396,18.094,152.949
C09926=1086.008,-42.011,-54.709,174.395,18.092,152.949
C09927=1086.002,-42.260,-54.697,174.393,18.090,152.949
C09928=1085.995,-42.510,-54.685,174.392,18.089,152.949
C09929=1085.990,-42.759,-54.672,174.390,18.087,152.949
C09930=1085.984,-43.009,-54.660,174.388,18.085,152.949
C09931=1085.977,-43.259,-54.649,174.387,18.084,152.948
C09932=1085.972,-43.508,-54.636,174.385,18.083,152.949
C09933=1085.965,-43.758,-54.624,174.384,18.081,152.949
C09934=1085.960,-44.008,-54.612,174.382,18.079,152.949
C09935=1085.954,-44.257,-54.600,174.381,18.078,152.948
C09936=1085.948,-44.507,-54.588,174.380,18.076,152.948
C09937=1085.942,-44.757,-54.576,174.378,18.075,152.948
C09938=1085.937,-45.006,-54.564,174.376,18.073,152.948
C09939=1085.930,-45.256,-54.552,174.375,18.071,152.948
C09940=1085.924,-45.506,-54.539,174.373,18.070,152.948
C09941=1085.918,-45.755,-54.528,174.372,18.068,152.948
C09942=1085.912,-46.005,-54.516,174.370,18.066,152.948
C09943=1085.906,-46.254,-54.504,174.369,18.065,152.948
C09944=1085.901,-46.504,-54.492,174.368,18.063,152.948
C09945=1085.895,-46.754,-54.480,174.366,18.062,152.948
C09946=1085.889,-47.003,-54.468,174.364,18.061,152.948
C09947=1085.883,-47.253,-54.456,174.363,18.059,152.948
C09948=1085.877,-47.502,-54.444,174.361,18.057,152.948
C09949=1085.871,-47.753,-54.432,174.359,18.055,152.948
C09950=1085.865,-48.002,-54.420,174.358,18.054,152.948
C09951=1085.859,-48.251,-54.408,174.357,18.052,152.948
C09952=1085.854,-48.502,-54.396,174.355,18.051,152.948
C09953=1085.847,-48.773,-54.383,174.354,18.049,152.948
C09954=1085.841,-49.045,-54.371,174.352,18.047,152.948
C09955=1085.834,-49.317,-54.358,174.350,18.046,152.948
C09956=1085.828,-49.590,-54.345,174.349,18.044,152.948
C09957=1085.822,-49.839,-54.333,174.347,18.042,152.948
C09958=1085.816,-50.089,-54.321,174.346,18.041,152.948
C09959=1085.811,-50.339,-54.309,174.345,18.039,152.948
C09960=1085.804,-50.588,-54.297,174.343,18.038,152.948
C09961=1085.799,-50.837,-54.285,174.341,18.037,152.948
C09962=1085.793,-51.087,-54.274,174.339,18.035,152.948
C09963=1085.786,-51.337,-54.262,174.338,18.033,152.948
C09964=1085.780,-51.587,-54.251,174.336,18.031,152.948
C09965=1085.774,-51.836,-54.238,174.335,18.030,152.948
C09966=1085.768,-52.086,-54.226,174.333,18.029,152.948
C09967=1085.762,-52.335,-54.215,174.332,18.027,152.948
C09968=1085.756,-52.585,-54.203,174.331,18.026,152.948
C09969=1085.750,-52.835,-54.192,174.329,18.024,152.948
C09970=1085.744,-53.084,-54.180,174.327,18.023,152.948
C09971=1085.738,-53.335,-54.168,174.326,18.022,152.948
C09972=1085.732,-53.584,-54.157,174.325,18.020,152.948
C09973=1085.725,-53.833,-54.145,174.323,18.018,152.948
C09974=1085.720,-54.083,-54.134,174.322,18.017,152.948
C09975=1085.714,-54.333,-54.121,174.320,18.016,152.948
C09976=1085.707,-54.583,-54.110,174.318,18.014,152.948
C09977=1085.701,-54.832,-54.098,174.317,18.012,152.948
C09978=1085.696,-55.082,-54.087,174.315,18.011,152.948
C09979=1085.690,-55.331,-54.075,174.314,18.010,152.948
C09980=1085.683,-55.581,-54.064,174.312,18.008,152.948
C09981=1085.677,-55.830,-54.052,174.311,18.006,152.948
C09982=1085.672,-56.081,-54.040,174.309,18.005,152.948
C09983=1085.666,-56.330,-54.029,174.308,18.004,152.948
C09984=1085.659,-56.580,-54.017,174.306,18.002,152.948
C09985=1085.653,-56.829,-54.006,174.305,18.001,152.948
C09986=1085.648,-57.079,-53.994,174.303,18.000,152.948
C09987=1085.641,-57.329,-53.983,174.302,17.998,152.948
C09988=1085.635,-57.578,-53.971,174.300,17.996,152.948
C09989=1085.629,-57.828,-53.960,174.299,17.995,152.948
C09990=1085.624,-58.078,-53.948,174.297,17.994,152.948
C09991=1085.617,-58.328,-53.937,174.296,17.992,152.948
C09992=1085.611,-58.577,-53.925,174.295,17.991,152.948
C09993=1085.605,-58.827,-53.914,174.293,17.989,152.948
C09994=1085.599,-59.076,-53.903,174.291,17.988,152.948
C09995=1085.593,-59.326,-53.890,174.289,17.986,152.948
C09996=1085.587,-59.576,-53.879,174.288,17.984,152.948
//INST
///DATE 2021/06/17 10:53
///ATTR SC,RW,RJ
////FRAME ROBOT
///GROUP1 RB1
NOP
MOVL C00000 V=800.0 PL=0
MOVL C00001 V=800.0 PL=0
MOVL C00002 V=800.0 PL=0
MOVL C00003 V=800.0 PL=0
MOVL C00004 V=800.0 PL=0
MOVL C00005 V=800.0 PL=0
MOVL C00006 V=800.0 PL=0
MOVL C00007 V=800.0 PL=0
MOVL C00008 V=800.0 PL=0
MOVL C00009 V=800.0 PL=0
MOVL C00010 V=800.0 PL=0
MOVL C00011 V=800.0 PL=0
MOVL C00012 V=800.0 PL=0
MOVL C00013 V=800.0 PL=0
MOVL C00014 V=800.0 PL=0
MOVL C00015 V=800.0 PL=0
MOVL C00016 V=800.0 PL=0
MOVL C00017 V=800.0 PL=0
MOVL C00018 V=800.0 PL=0
MOVL C00019 V=800.0 PL=0
MOVL C00020 V=800.0 PL=0
MOVL C00021 V=800.0 PL=0
MOVL C00022 V=800.0 PL=0
MOVL C00023 V=800.0 PL=0
MOVL C00024 V=800.0 PL=0
MOVL C00025 V=800.0 PL=0
MOVL C00026 V=800.0 PL=0
MOVL C00027 V=800.0 PL=0
MOVL C00028 V=800.0 PL=0
MOVL C00029 V=800.0 PL=0
MOVL C00030 V=800.0 PL=0
MOVL C00031 V=800.0 PL=0
MOVL C00032 V=800.0 PL=0
MOVL C00033 V=800.0 PL=0
MOVL C00034 V=800.0 PL=0
MOVL C00035 V=800.0 PL=0
MOVL C00036 V=800.0 PL=0
MOVL C00037 V=800.0 PL=0
MOVL C00038 V=800.0 PL=0
MOVL C00039 V=800.0 PL=0
MOVL C00040 V=800.0 PL=0
MOVL C00041 V=800.0 PL=0
MOVL C00042 V=800.0 PL=0
MOVL C00043 V=800.0 PL=0
MOVL C00044 V=800.0 PL=0
MOVL C00045 V=800.0 PL=0
MOVL C00046 V=800.0 PL=0
MOVL C00047 V=800.0 PL=0
MOVL C00048 V=800.0 PL=0
MOVL C00049 V=800.0 PL=0
MOVL C00050 V=800.0 PL=0
MOVL C00051 V=800.0 PL=0
MOVL C00052 V=800.0 PL=0
MOVL C00053 V=800.0 PL=0
MOVL C00054 V=800.0 PL=0
MOVL C00055 V=800.0 PL=0
MOVL C00056 V=800.0 PL=0
MOVL C00057 V=800.0 PL=0
MOVL C00058 V=800.0 PL=0
MOVL C00059 V=800.0 PL=0
MOVL C00060 V=800.0 PL=0
MOVL C00061 V=800.0 PL=0
MOVL C00062 V=800.0 PL=0
MOVL C00063 V=800.0 PL=0
MOVL C00064 V=800.0 PL=0
MOVL C00065 V=800.0 PL=0
MOVL C00066 V=800.0 PL=0
MOVL C00067 V=800.0 PL=0
MOVL C00068 V=800.0 PL=0
MOVL C00069 V=800.0 PL=0
MOVL C00070 V=800.0 PL=0
MOVL C00071 V=800.0 PL=0
MOVL C00072 V=800.0 PL=0
MOVL C00073 V=800.0 PL=0
MOVL C00074 V=800.0 PL=0
MOVL C00075 V=800.0 PL=0
MOVL C00076 V=800.0 PL=0
MOVL C00077 V=800.0 PL=0
MOVL C00078 V=800.0 PL=0
MOVL C00079 V=800.0 PL=0
MOVL C00080 V=800.0 PL=0
MOVL C00081 V=800.0 PL=0
MOVL C00082 V=800.0 PL=0
MOVL C00083 V=800.0 PL=0
MOVL C00084 V=800.0 PL=0
MOVL C00085 V=800.0 PL=0
MOVL C00086 V=800.0 PL=0
MOVL C00087 V=800.0 PL=0
MOVL C00088 V=800.0 PL=0
MOVL C00089 V=800.0 PL=0
MOVL C00090 V=800.0 PL=0
MOVL C00091 V=800.0 PL=0
MOVL C00092 V=800.0 PL=0
MOVL C00093 V=800.0 PL=0
MOVL C00094 V=800.0 PL=0
MOVL C00095 V=800.0 PL=0
MOVL C00096 V=800.0 PL=0
MOVL C00097 V=800.0 PL=0
MOVL C00098 V=800.0 PL=0
MOVL C00099 V=800.0 PL=0
MOVL C00100 V=800.0 PL=0
MOVL C00101 V=800.0 PL=0
MOVL C00102 V=800.0 PL=0
MOVL C00103 V=800.0 PL=0
MOVL C00104 V=800.0 PL=0
MOVL C00105 V=800.0 PL=0
MOVL C00106 V=800.0 PL=0
MOVL C00107 V=800.0 PL=0
MOVL C00108 V=800.0 PL=0
MOVL C00109 V=800.0 PL=0
MOVL C00110 V=800.0 PL=0
MOVL C00111 V=800.0 PL=0
MOVL C00112 V=800.0 PL=0
MOVL C00113 V=800.0 PL=0
MOVL C00114 V=800.0 PL=0
MOVL C00115 V=800.0 PL=0
MOVL C00116 V=800.0 PL=0
MOVL C00117 V=800.0 PL=0
MOVL C00118 V=800.0 PL=0
MOVL C00119 V=800.0 PL=0
MOVL C00120 V=800.0 PL=0
MOVL C00121 V=800.0 PL=0
MOVL C00122 V=800.0 PL=0
MOVL C00123 V=800.0 PL=0
MOVL C00124 V=800.0 PL=0
MOVL C00125 V=800.0 PL=0
MOVL C00126 V=800.0 PL=0
MOVL C00127 V=800.0 PL=0
MOVL C00128 V=800.0 PL=0
MOVL C00129 V=800.0 PL=0
MOVL C00130 V=800.0 PL=0
MOVL C00131 V=800.0 PL=0
MOVL C00132 V=800.0 PL=0
MOVL C00133 V=800.0 PL=0
MOVL C00134 V=800.0 PL=0
MOVL C00135 V=800.0 PL=0
MOVL C00136 V=800.0 PL=0
MOVL C00137 V=800.0 PL=0
MOVL C00138 V=800.0 PL=0
MOVL C00139 V=800.0 PL=0
MOVL C00140 V=800.0 PL=0
MOVL C00141 V=800.0 PL=0
MOVL C00142 V=800.0 PL=0
MOVL C00143 V=800.0 PL=0
MOVL C00144 V=800.0 PL=0
MOVL C00145 V=800.0 PL=0
MOVL C00146 V=800.0 PL=0
MOVL C00147 V=800.0 PL=0
MOVL C00148 V=800.0 PL=0
MOVL C00149 V=800.0 PL=0
MOVL C00150 V=800.0 PL=0
MOVL C00151 V=800.0 PL=0
MOVL C00152 V=800.0 PL=0
MOVL C00153 V=800.0 PL=0
MOVL C00154 V=800.0 PL=0
MOVL C00155 V=800.0 PL=0
MOVL C00156 V=800.0 PL=0
MOVL C00157 V=800.0 PL=0
MOVL C00158 V=800.0 PL=0
MOVL C00159 V=800.0 PL=0
MOVL C00160 V=800.0 PL=0
MOVL C00161 V=800.0 PL=0
MOVL C00162 V=800.0 PL=0
MOVL C00163 V=800.0 PL=0
MOVL C00164 V=800.0 PL=0
MOVL C00165 V=800.0 PL=0
MOVL C00166 V=800.0 PL=0
MOVL C00167 V=800.0 PL=0
MOVL C00168 V=800.0 PL=0
MOVL C00169 V=800.0 PL=0
MOVL C00170 V=800.0 PL=0
MOVL C00171 V=800.0 PL=0
MOVL C00172 V=800.0 PL=0
MOVL C00173 V=800.0 PL=0
MOVL C00174 V=800.0 PL=0
MOVL C00175 V=800.0 PL=0
MOVL C00176 V=800.0 PL=0
MOVL C00177 V=800.0 PL=0
MOVL C00178 V=800.0 PL=0
MOVL C00179 V=800.0 PL=0
MOVL C00180 V=800.0 PL=0
MOVL C00181 V=800.0 PL=0
MOVL C00182 V=800.0 PL=0
MOVL C00183 V=800.0 PL=0
MOVL C00184 V=800.0 PL=0
MOVL C00185 V=800.0 PL=0
MOVL C00186 V=800.0 PL=0
MOVL C00187 V=800.0 PL=0
MOVL C00188 V=800.0 PL=0
MOVL C00189 V=800.0 PL=0
MOVL C00190 V=800.0 PL=0
MOVL C00191 V=800.0 PL=0
MOVL C00192 V=800.0 PL=0
MOVL C00193 V=800.0 PL=0
MOVL C00194 V=800.0 PL=0
MOVL C00195 V=800.0 PL=0
MOVL C00196 V=800.0 PL=0
MOVL C00197 V=800.0 PL=0
MOVL C00198 V=800.0 PL=0
MOVL C00199 V=800.0 PL=0
MOVL C00200 V=800.0 PL=0
MOVL C00201 V=800.0 PL=0
MOVL C00202 V=800.0 PL=0
MOVL C00203 V=800.0 PL=0
MOVL C00204 V=800.0 PL=0
MOVL C00205 V=800.0 PL=0
MOVL C00206 V=800.0 PL=0
MOVL C00207 V=800.0 PL=0
MOVL C00208 V=800.0 PL=0
MOVL C00209 V=800.0 PL=0
MOVL C00210 V=800.0 PL=0
MOVL C00211 V=800.0 PL=0
MOVL C00212 V=800.0 PL=0
MOVL C00213 V=800.0 PL=0
MOVL C00214 V=800.0 PL=0
MOVL C00215 V=800.0 PL=0
MOVL C00216 V=800.0 PL=0
MOVL C00217 V=800.0 PL=0
MOVL C00218 V=800.0 PL=0
MOVL C00219 V=800.0 PL=0
MOVL C00220 V=800.0 PL=0
MOVL C00221 V=800.0 PL=0
MOVL C00222 V=800.0 PL=0
MOVL C00223 V=800.0 PL=0
MOVL C00224 V=800.0 PL=0
MOVL C00225 V=800.0 PL=0
MOVL C00226 V=800.0 PL=0
MOVL C00227 V=800.0 PL=0
MOVL C00228 V=800.0 PL=0
MOVL C00229 V=800.0 PL=0
MOVL C00230 V=800.0 PL=0
MOVL C00231 V=800.0 PL=0
MOVL C00232 V=800.0 PL=0
MOVL C00233 V=800.0 PL=0
MOVL C00234 V=800.0 PL=0
MOVL C00235 V=800.0 PL=0
MOVL C00236 V=800.0 PL=0
MOVL C00237 V=800.0 PL=0
MOVL C00238 V=800.0 PL=0
MOVL C00239 V=800.0 PL=0
MOVL C00240 V=800.0 PL=0
MOVL C00241 V=800.0 PL=0
MOVL C00242 V=800.0 PL=0
MOVL C00243 V=800.0 PL=0
MOVL C00244 V=800.0 PL=0
MOVL C00245 V=800.0 PL=0
MOVL C00246 V=800.0 PL=0
MOVL C00247 V=800.0 PL=0
MOVL C00248 V=800.0 PL=0
MOVL C00249 V=800.0 PL=0
MOVL C00250 V=800.0 PL=0
MOVL C00251 V=800.0 PL=0
MOVL C00252 V=800.0 PL=0
MOVL C00253 V=800.0 PL=0
MOVL C00254 V=800.0 PL=0
MOVL C00255 V=800.0 PL=0
MOVL C00256 V=800.0 PL=0
MOVL C00257 V=800.0 PL=0
MOVL C00258 V=800.0 PL=0
MOVL C00259 V=800.0 PL=0
MOVL C00260 V=800.0 PL=0
MOVL C00261 V=800.0 PL=0
MOVL C00262 V=800.0 PL=0
MOVL C00263 V=800.0 PL=0
MOVL C00264 V=800.0 PL=0
MOVL C00265 V=800.0 PL=0
MOVL C00266 V=800.0 PL=0
MOVL C00267 V=800.0 PL=0
MOVL C00268 V=800.0 PL=0
MOVL C00269 V=800.0 PL=0
MOVL C00270 V=800.0 PL=0
MOVL C00271 V=800.0 PL=0
MOVL C00272 V=800.0 PL=0
MOVL C00273 V=800.0 PL=0
MOVL C00274 V=800.0 PL=0
MOVL C00275 V=800.0 PL=0
MOVL C00276 V=800.0 PL=0
MOVL C00277 V=800.0 PL=0
MOVL C00278 V=800.0 PL=0
MOVL C00279 V=800.0 PL=0
MOVL C00280 V=800.0 PL=0
MOVL C00281 V=800.0 PL=0
MOVL C00282 V=800.0 PL=0
MOVL C00283 V=800.0 PL=0
MOVL C00284 V=800.0 PL=0
MOVL C00285 V=800.0 PL=0
MOVL C00286 V=800.0 PL=0
MOVL C00287 V=800.0 PL=0
MOVL C00288 V=800.0 PL=0
MOVL C00289 V=800.0 PL=0
MOVL C00290 V=800.0 PL=0
MOVL C00291 V=800.0 PL=0
MOVL C00292 V=800.0 PL=0
MOVL C00293 V=800.0 PL=0
MOVL C00294 V=800.0 PL=0
MOVL C00295 V=800.0 PL=0
MOVL C00296 V=800.0 PL=0
MOVL C00297 V=800.0 PL=0
MOVL C00298 V=800.0 PL=0
MOVL C00299 V=800.0 PL=0
MOVL C00300 V=800.0 PL=0
MOVL C00301 V=800.0 PL=0
MOVL C00302 V=800.0 PL=0
MOVL C00303 V=800.0 PL=0
MOVL C00304 V=800.0 PL=0
MOVL C00305 V=800.0 PL=0
MOVL C00306 V=800.0 PL=0
MOVL C00307 V=800.0 PL=0
MOVL C00308 V=800.0 PL=0
MOVL C00309 V=800.0 PL=0
MOVL C00310 V=800.0 PL=0
MOVL C00311 V=800.0 PL=0
MOVL C00312 V=800.0 PL=0
MOVL C00313 V=800.0 PL=0
MOVL C00314 V=800.0 PL=0
MOVL C00315 V=800.0 PL=0
MOVL C00316 V=800.0 PL=0
MOVL C00317 V=800.0 PL=0
MOVL C00318 V=800.0 PL=0
MOVL C00319 V=800.0 PL=0
MOVL C00320 V=800.0 PL=0
MOVL C00321 V=800.0 PL=0
MOVL C00322 V=800.0 PL=0
MOVL C00323 V=800.0 PL=0
MOVL C00324 V=800.0 PL=0
MOVL C00325 V=800.0 PL=0
MOVL C00326 V=800.0 PL=0
MOVL C00327 V=800.0 PL=0
MOVL C00328 V=800.0 PL=0
MOVL C00329 V=800.0 PL=0
MOVL C00330 V=800.0 PL=0
MOVL C00331 V=800.0 PL=0
MOVL C00332 V=800.0 PL=0
MOVL C00333 V=800.0 PL=0
MOVL C00334 V=800.0 PL=0
MOVL C00335 V=800.0 PL=0
MOVL C00336 V=800.0 PL=0
MOVL C00337 V=800.0 PL=0
MOVL C00338 V=800.0 PL=0
MOVL C00339 V=800.0 PL=0
MOVL C00340 V=800.0 PL=0
MOVL C00341 V=800.0 PL=0
MOVL C00342 V=800.0 PL=0
MOVL C00343 V=800.0 PL=0
MOVL C00344 V=800.0 PL=0
MOVL C00345 V=800.0 PL=0
MOVL C00346 V=800.0 PL=0
MOVL C00347 V=800.0 PL=0
MOVL C00348 V=800.0 PL=0
MOVL C00349 V=800.0 PL=0
MOVL C00350 V=800.0 PL=0
MOVL C00351 V=800.0 PL=0
MOVL C00352 V=800.0 PL=0
MOVL C00353 V=800.0 PL=0
MOVL C00354 V=800.0 PL=0
MOVL C00355 V=800.0 PL=0
MOVL C00356 V=800.0 PL=0
MOVL C00357 V=800.0 PL=0
MOVL C00358 V=800.0 PL=0
MOVL C00359 V=800.0 PL=0
MOVL C00360 V=800.0 PL=0
MOVL C00361 V=800.0 PL=0
MOVL C00362 V=800.0 PL=0
MOVL C00363 V=800.0 PL=0
MOVL C00364 V=800.0 PL=0
MOVL C00365 V=800.0 PL=0
MOVL C00366 V=800.0 PL=0
MOVL C00367 V=800.0 PL=0
MOVL C00368 V=800.0 PL=0
MOVL C00369 V=800.0 PL=0
MOVL C00370 V=800.0 PL=0
MOVL C00371 V=800.0 PL=0
MOVL C00372 V=800.0 PL=0
MOVL C00373 V=800.0 PL=0
MOVL C00374 V=800.0 PL=0
MOVL C00375 V=800.0 PL=0
MOVL C00376 V=800.0 PL=0
MOVL C00377 V=800.0 PL=0
MOVL C00378 V=800.0 PL=0
MOVL C00379 V=800.0 PL=0
MOVL C00380 V=800.0 PL=0
MOVL C00381 V=800.0 PL=0
MOVL C00382 V=800.0 PL=0
MOVL C00383 V=800.0 PL=0
MOVL C00384 V=800.0 PL=0
MOVL C00385 V=800.0 PL=0
MOVL C00386 V=800.0 PL=0
MOVL C00387 V=800.0 PL=0
MOVL C00388 V=800.0 PL=0
MOVL C00389 V=800.0 PL=0
MOVL C00390 V=800.0 PL=0
MOVL C00391 V=800.0 PL=0
MOVL C00392 V=800.0 PL=0
MOVL C00393 V=800.0 PL=0
MOVL C00394 V=800.0 PL=0
MOVL C00395 V=800.0 PL=0
MOVL C00396 V=800.0 PL=0
MOVL C00397 V=800.0 PL=0
MOVL C00398 V=800.0 PL=0
MOVL C00399 V=800.0 PL=0
MOVL C00400 V=800.0 PL=0
MOVL C00401 V=800.0 PL=0
MOVL C00402 V=800.0 PL=0
MOVL C00403 V=800.0 PL=0
MOVL C00404 V=800.0 PL=0
MOVL C00405 V=800.0 PL=0
MOVL C00406 V=800.0 PL=0
MOVL C00407 V=800.0 PL=0
MOVL C00408 V=800.0 PL=0
MOVL C00409 V=800.0 PL=0
MOVL C00410 V=800.0 PL=0
MOVL C00411 V=800.0 PL=0
MOVL C00412 V=800.0 PL=0
MOVL C00413 V=800.0 PL=0
MOVL C00414 V=800.0 PL=0
MOVL C00415 V=800.0 PL=0
MOVL C00416 V=800.0 PL=0
MOVL C00417 V=800.0 PL=0
MOVL C00418 V=800.0 PL=0
MOVL C00419 V=800.0 PL=0
MOVL C00420 V=800.0 PL=0
MOVL C00421 V=800.0 PL=0
MOVL C00422 V=800.0 PL=0
MOVL C00423 V=800.0 PL=0
MOVL C00424 V=800.0 PL=0
MOVL C00425 V=800.0 PL=0
MOVL C00426 V=800.0 PL=0
MOVL C00427 V=800.0 PL=0
MOVL C00428 V=800.0 PL=0
MOVL C00429 V=800.0 PL=0
MOVL C00430 V=800.0 PL=0
MOVL C00431 V=800.0 PL=0
MOVL C00432 V=800.0 PL=0
MOVL C00433 V=800.0 PL=0
MOVL C00434 V=800.0 PL=0
MOVL C00435 V=800.0 PL=0
MOVL C00436 V=800.0 PL=0
MOVL C00437 V=800.0 PL=0
MOVL C00438 V=800.0 PL=0
MOVL C00439 V=800.0 PL=0
MOVL C00440 V=800.0 PL=0
MOVL C00441 V=800.0 PL=0
MOVL C00442 V=800.0 PL=0
MOVL C00443 V=800.0 PL=0
MOVL C00444 V=800.0 PL=0
MOVL C00445 V=800.0 PL=0
MOVL C00446 V=800.0 PL=0
MOVL C00447 V=800.0 PL=0
MOVL C00448 V=800.0 PL=0
MOVL C00449 V=800.0 PL=0
MOVL C00450 V=800.0 PL=0
MOVL C00451 V=800.0 PL=0
MOVL C00452 V=800.0 PL=0
MOVL C00453 V=800.0 PL=0
MOVL C00454 V=800.0 PL=0
MOVL C00455 V=800.0 PL=0
MOVL C00456 V=800.0 PL=0
MOVL C00457 V=800.0 PL=0
MOVL C00458 V=800.0 PL=0
MOVL C00459 V=800.0 PL=0
MOVL C00460 V=800.0 PL=0
MOVL C00461 V=800.0 PL=0
MOVL C00462 V=800.0 PL=0
MOVL C00463 V=800.0 PL=0
MOVL C00464 V=800.0 PL=0
MOVL C00465 V=800.0 PL=0
MOVL C00466 V=800.0 PL=0
MOVL C00467 V=800.0 PL=0
MOVL C00468 V=800.0 PL=0
MOVL C00469 V=800.0 PL=0
MOVL C00470 V=800.0 PL=0
MOVL C00471 V=800.0 PL=0
MOVL C00472 V=800.0 PL=0
MOVL C00473 V=800.0 PL=0
MOVL C00474 V=800.0 PL=0
MOVL C00475 V=800.0 PL=0
MOVL C00476 V=800.0 PL=0
MOVL C00477 V=800.0 PL=0
MOVL C00478 V=800.0 PL=0
MOVL C00479 V=800.0 PL=0
MOVL C00480 V=800.0 PL=0
MOVL C00481 V=800.0 PL=0
MOVL C00482 V=800.0 PL=0
MOVL C00483 V=800.0 PL=0
MOVL C00484 V=800.0 PL=0
MOVL C00485 V=800.0 PL=0
MOVL C00486 V=800.0 PL=0
MOVL C00487 V=800.0 PL=0
MOVL C00488 V=800.0 PL=0
MOVL C00489 V=800.0 PL=0
MOVL C00490 V=800.0 PL=0
MOVL C00491 V=800.0 PL=0
MOVL C00492 V=800.0 PL=0
MOVL C00493 V=800.0 PL=0
MOVL C00494 V=800.0 PL=0
MOVL C00495 V=800.0 PL=0
MOVL C00496 V=800.0 PL=0
MOVL C00497 V=800.0 PL=0
MOVL C00498 V=800.0 PL=0
MOVL C00499 V=800.0 PL=0
MOVL C00500 V=800.0 PL=0
MOVL C00501 V=800.0 PL=0
MOVL C00502 V=800.0 PL=0
MOVL C00503 V=800.0 PL=0
MOVL C00504 V=800.0 PL=0
MOVL C00505 V=800.0 PL=0
MOVL C00506 V=800.0 PL=0
MOVL C00507 V=800.0 PL=0
MOVL C00508 V=800.0 PL=0
MOVL C00509 V=800.0 PL=0
MOVL C00510 V=800.0 PL=0
MOVL C00511 V=800.0 PL=0
MOVL C00512 V=800.0 PL=0
MOVL C00513 V=800.0 PL=0
MOVL C00514 V=800.0 PL=0
MOVL C00515 V=800.0 PL=0
MOVL C00516 V=800.0 PL=0
MOVL C00517 V=800.0 PL=0
MOVL C00518 V=800.0 PL=0
MOVL C00519 V=800.0 PL=0
MOVL C00520 V=800.0 PL=0
MOVL C00521 V=800.0 PL=0
MOVL C00522 V=800.0 PL=0
MOVL C00523 V=800.0 PL=0
MOVL C00524 V=800.0 PL=0
MOVL C00525 V=800.0 PL=0
MOVL C00526 V=800.0 PL=0
MOVL C00527 V=800.0 PL=0
MOVL C00528 V=800.0 PL=0
MOVL C00529 V=800.0 PL=0
MOVL C00530 V=800.0 PL=0
MOVL C00531 V=800.0 PL=0
MOVL C00532 V=800.0 PL=0
MOVL C00533 V=800.0 PL=0
MOVL C00534 V=800.0 PL=0
MOVL C00535 V=800.0 PL=0
MOVL C00536 V=800.0 PL=0
MOVL C00537 V=800.0 PL=0
MOVL C00538 V=800.0 PL=0
MOVL C00539 V=800.0 PL=0
MOVL C00540 V=800.0 PL=0
MOVL C00541 V=800.0 PL=0
MOVL C00542 V=800.0 PL=0
MOVL C00543 V=800.0 PL=0
MOVL C00544 V=800.0 PL=0
MOVL C00545 V=800.0 PL=0
MOVL C00546 V=800.0 PL=0
MOVL C00547 V=800.0 PL=0
MOVL C00548 V=800.0 PL=0
MOVL C00549 V=800.0 PL=0
MOVL C00550 V=800.0 PL=0
MOVL C00551 V=800.0 PL=0
MOVL C00552 V=800.0 PL=0
MOVL C00553 V=800.0 PL=0
MOVL C00554 V=800.0 PL=0
MOVL C00555 V=800.0 PL=0
MOVL C00556 V=800.0 PL=0
MOVL C00557 V=800.0 PL=0
MOVL C00558 V=800.0 PL=0
MOVL C00559 V=800.0 PL=0
MOVL C00560 V=800.0 PL=0
MOVL C00561 V=800.0 PL=0
MOVL C00562 V=800.0 PL=0
MOVL C00563 V=800.0 PL=0
MOVL C00564 V=800.0 PL=0
MOVL C00565 V=800.0 PL=0
MOVL C00566 V=800.0 PL=0
MOVL C00567 V=800.0 PL=0
MOVL C00568 V=800.0 PL=0
MOVL C00569 V=800.0 PL=0
MOVL C00570 V=800.0 PL=0
MOVL C00571 V=800.0 PL=0
MOVL C00572 V=800.0 PL=0
MOVL C00573 V=800.0 PL=0
MOVL C00574 V=800.0 PL=0
MOVL C00575 V=800.0 PL=0
MOVL C00576 V=800.0 PL=0
MOVL C00577 V=800.0 PL=0
MOVL C00578 V=800.0 PL=0
MOVL C00579 V=800.0 PL=0
MOVL C00580 V=800.0 PL=0
MOVL C00581 V=800.0 PL=0
MOVL C00582 V=800.0 PL=0
MOVL C00583 V=800.0 PL=0
MOVL C00584 V=800.0 PL=0
MOVL C00585 V=800.0 PL=0
MOVL C00586 V=800.0 PL=0
MOVL C00587 V=800.0 PL=0
MOVL C00588 V=800.0 PL=0
MOVL C00589 V=800.0 PL=0
MOVL C00590 V=800.0 PL=0
MOVL C00591 V=800.0 PL=0
MOVL C00592 V=800.0 PL=0
MOVL C00593 V=800.0 PL=0
MOVL C00594 V=800.0 PL=0
MOVL C00595 V=800.0 PL=0
MOVL C00596 V=800.0 PL=0
MOVL C00597 V=800.0 PL=0
MOVL C00598 V=800.0 PL=0
MOVL C00599 V=800.0 PL=0
MOVL C00600 V=800.0 PL=0
MOVL C00601 V=800.0 PL=0
MOVL C00602 V=800.0 PL=0
MOVL C00603 V=800.0 PL=0
MOVL C00604 V=800.0 PL=0
MOVL C00605 V=800.0 PL=0
MOVL C00606 V=800.0 PL=0
MOVL C00607 V=800.0 PL=0
MOVL C00608 V=800.0 PL=0
MOVL C00609 V=800.0 PL=0
MOVL C00610 V=800.0 PL=0
MOVL C00611 V=800.0 PL=0
MOVL C00612 V=800.0 PL=0
MOVL C00613 V=800.0 PL=0
MOVL C00614 V=800.0 PL=0
MOVL C00615 V=800.0 PL=0
MOVL C00616 V=800.0 PL=0
MOVL C00617 V=800.0 PL=0
MOVL C00618 V=800.0 PL=0
MOVL C00619 V=800.0 PL=0
MOVL C00620 V=800.0 PL=0
MOVL C00621 V=800.0 PL=0
MOVL C00622 V=800.0 PL=0
MOVL C00623 V=800.0 PL=0
MOVL C00624 V=800.0 PL=0
MOVL C00625 V=800.0 PL=0
MOVL C00626 V=800.0 PL=0
MOVL C00627 V=800.0 PL=0
MOVL C00628 V=800.0 PL=0
MOVL C00629 V=800.0 PL=0
MOVL C00630 V=800.0 PL=0
MOVL C00631 V=800.0 PL=0
MOVL C00632 V=800.0 PL=0
MOVL C00633 V=800.0 PL=0
MOVL C00634 V=800.0 PL=0
MOVL C00635 V=800.0 PL=0
MOVL C00636 V=800.0 PL=0
MOVL C00637 V=800.0 PL=0
MOVL C00638 V=800.0 PL=0
MOVL C00639 V=800.0 PL=0
MOVL C00640 V=800.0 PL=0
MOVL C00641 V=800.0 PL=0
MOVL C00642 V=800.0 PL=0
MOVL C00643 V=800.0 PL=0
MOVL C00644 V=800.0 PL=0
MOVL C00645 V=800.0 PL=0
MOVL C00646 V=800.0 PL=0
MOVL C00647 V=800.0 PL=0
MOVL C00648 V=800.0 PL=0
MOVL C00649 V=800.0 PL=0
MOVL C00650 V=800.0 PL=0
MOVL C00651 V=800.0 PL=0
MOVL C00652 V=800.0 PL=0
MOVL C00653 V=800.0 PL=0
MOVL C00654 V=800.0 PL=0
MOVL C00655 V=800.0 PL=0
MOVL C00656 V=800.0 PL=0
MOVL C00657 V=800.0 PL=0
MOVL C00658 V=800.0 PL=0
MOVL C00659 V=800.0 PL=0
MOVL C00660 V=800.0 PL=0
MOVL C00661 V=800.0 PL=0
MOVL C00662 V=800.0 PL=0
MOVL C00663 V=800.0 PL=0
MOVL C00664 V=800.0 PL=0
MOVL C00665 V=800.0 PL=0
MOVL C00666 V=800.0 PL=0
MOVL C00667 V=800.0 PL=0
MOVL C00668 V=800.0 PL=0
MOVL C00669 V=800.0 PL=0
MOVL C00670 V=800.0 PL=0
MOVL C00671 V=800.0 PL=0
MOVL C00672 V=800.0 PL=0
MOVL C00673 V=800.0 PL=0
MOVL C00674 V=800.0 PL=0
MOVL C00675 V=800.0 PL=0
MOVL C00676 V=800.0 PL=0
MOVL C00677 V=800.0 PL=0
MOVL C00678 V=800.0 PL=0
MOVL C00679 V=800.0 PL=0
MOVL C00680 V=800.0 PL=0
MOVL C00681 V=800.0 PL=0
MOVL C00682 V=800.0 PL=0
MOVL C00683 V=800.0 PL=0
MOVL C00684 V=800.0 PL=0
MOVL C00685 V=800.0 PL=0
MOVL C00686 V=800.0 PL=0
MOVL C00687 V=800.0 PL=0
MOVL C00688 V=800.0 PL=0
MOVL C00689 V=800.0 PL=0
MOVL C00690 V=800.0 PL=0
MOVL C00691 V=800.0 PL=0
MOVL C00692 V=800.0 PL=0
MOVL C00693 V=800.0 PL=0
MOVL C00694 V=800.0 PL=0
MOVL C00695 V=800.0 PL=0
MOVL C00696 V=800.0 PL=0
MOVL C00697 V=800.0 PL=0
MOVL C00698 V=800.0 PL=0
MOVL C00699 V=800.0 PL=0
MOVL C00700 V=800.0 PL=0
MOVL C00701 V=800.0 PL=0
MOVL C00702 V=800.0 PL=0
MOVL C00703 V=800.0 PL=0
MOVL C00704 V=800.0 PL=0
MOVL C00705 V=800.0 PL=0
MOVL C00706 V=800.0 PL=0
MOVL C00707 V=800.0 PL=0
MOVL C00708 V=800.0 PL=0
MOVL C00709 V=800.0 PL=0
MOVL C00710 V=800.0 PL=0
MOVL C00711 V=800.0 PL=0
MOVL C00712 V=800.0 PL=0
MOVL C00713 V=800.0 PL=0
MOVL C00714 V=800.0 PL=0
MOVL C00715 V=800.0 PL=0
MOVL C00716 V=800.0 PL=0
MOVL C00717 V=800.0 PL=0
MOVL C00718 V=800.0 PL=0
MOVL C00719 V=800.0 PL=0
MOVL C00720 V=800.0 PL=0
MOVL C00721 V=800.0 PL=0
MOVL C00722 V=800.0 PL=0
MOVL C00723 V=800.0 PL=0
MOVL C00724 V=800.0 PL=0
MOVL C00725 V=800.0 PL=0
MOVL C00726 V=800.0 PL=0
MOVL C00727 V=800.0 PL=0
MOVL C00728 V=800.0 PL=0
MOVL C00729 V=800.0 PL=0
MOVL C00730 V=800.0 PL=0
MOVL C00731 V=800.0 PL=0
MOVL C00732 V=800.0 PL=0
MOVL C00733 V=800.0 PL=0
MOVL C00734 V=800.0 PL=0
MOVL C00735 V=800.0 PL=0
MOVL C00736 V=800.0 PL=0
MOVL C00737 V=800.0 PL=0
MOVL C00738 V=800.0 PL=0
MOVL C00739 V=800.0 PL=0
MOVL C00740 V=800.0 PL=0
MOVL C00741 V=800.0 PL=0
MOVL C00742 V=800.0 PL=0
MOVL C00743 V=800.0 PL=0
MOVL C00744 V=800.0 PL=0
MOVL C00745 V=800.0 PL=0
MOVL C00746 V=800.0 PL=0
MOVL C00747 V=800.0 PL=0
MOVL C00748 V=800.0 PL=0
MOVL C00749 V=800.0 PL=0
MOVL C00750 V=800.0 PL=0
MOVL C00751 V=800.0 PL=0
MOVL C00752 V=800.0 PL=0
MOVL C00753 V=800.0 PL=0
MOVL C00754 V=800.0 PL=0
MOVL C00755 V=800.0 PL=0
MOVL C00756 V=800.0 PL=0
MOVL C00757 V=800.0 PL=0
MOVL C00758 V=800.0 PL=0
MOVL C00759 V=800.0 PL=0
MOVL C00760 V=800.0 PL=0
MOVL C00761 V=800.0 PL=0
MOVL C00762 V=800.0 PL=0
MOVL C00763 V=800.0 PL=0
MOVL C00764 V=800.0 PL=0
MOVL C00765 V=800.0 PL=0
MOVL C00766 V=800.0 PL=0
MOVL C00767 V=800.0 PL=0
MOVL C00768 V=800.0 PL=0
MOVL C00769 V=800.0 PL=0
MOVL C00770 V=800.0 PL=0
MOVL C00771 V=800.0 PL=0
MOVL C00772 V=800.0 PL=0
MOVL C00773 V=800.0 PL=0
MOVL C00774 V=800.0 PL=0
MOVL C00775 V=800.0 PL=0
MOVL C00776 V=800.0 PL=0
MOVL C00777 V=800.0 PL=0
MOVL C00778 V=800.0 PL=0
MOVL C00779 V=800.0 PL=0
MOVL C00780 V=800.0 PL=0
MOVL C00781 V=800.0 PL=0
MOVL C00782 V=800.0 PL=0
MOVL C00783 V=800.0 PL=0
MOVL C00784 V=800.0 PL=0
MOVL C00785 V=800.0 PL=0
MOVL C00786 V=800.0 PL=0
MOVL C00787 V=800.0 PL=0
MOVL C00788 V=800.0 PL=0
MOVL C00789 V=800.0 PL=0
MOVL C00790 V=800.0 PL=0
MOVL C00791 V=800.0 PL=0
MOVL C00792 V=800.0 PL=0
MOVL C00793 V=800.0 PL=0
MOVL C00794 V=800.0 PL=0
MOVL C00795 V=800.0 PL=0
MOVL C00796 V=800.0 PL=0
MOVL C00797 V=800.0 PL=0
MOVL C00798 V=800.0 PL=0
MOVL C00799 V=800.0 PL=0
MOVL C00800 V=800.0 PL=0
MOVL C00801 V=800.0 PL=0
MOVL C00802 V=800.0 PL=0
MOVL C00803 V=800.0 PL=0
MOVL C00804 V=800.0 PL=0
MOVL C00805 V=800.0 PL=0
MOVL C00806 V=800.0 PL=0
MOVL C00807 V=800.0 PL=0
MOVL C00808 V=800.0 PL=0
MOVL C00809 V=800.0 PL=0
MOVL C00810 V=800.0 PL=0
MOVL C00811 V=800.0 PL=0
MOVL C00812 V=800.0 PL=0
MOVL C00813 V=800.0 PL=0
MOVL C00814 V=800.0 PL=0
MOVL C00815 V=800.0 PL=0
MOVL C00816 V=800.0 PL=0
MOVL C00817 V=800.0 PL=0
MOVL C00818 V=800.0 PL=0
MOVL C00819 V=800.0 PL=0
MOVL C00820 V=800.0 PL=0
MOVL C00821 V=800.0 PL=0
MOVL C00822 V=800.0 PL=0
MOVL C00823 V=800.0 PL=0
MOVL C00824 V=800.0 PL=0
MOVL C00825 V=800.0 PL=0
MOVL C00826 V=800.0 PL=0
MOVL C00827 V=800.0 PL=0
MOVL C00828 V=800.0 PL=0
MOVL C00829 V=800.0 PL=0
MOVL C00830 V=800.0 PL=0
MOVL C00831 V=800.0 PL=0
MOVL C00832 V=800.0 PL=0
MOVL C00833 V=800.0 PL=0
MOVL C00834 V=800.0 PL=0
MOVL C00835 V=800.0 PL=0
MOVL C00836 V=800.0 PL=0
MOVL C00837 V=800.0 PL=0
MOVL C00838 V=800.0 PL=0
MOVL C00839 V=800.0 PL=0
MOVL C00840 V=800.0 PL=0
MOVL C00841 V=800.0 PL=0
MOVL C00842 V=800.0 PL=0
MOVL C00843 V=800.0 PL=0
MOVL C00844 V=800.0 PL=0
MOVL C00845 V=800.0 PL=0
MOVL C00846 V=800.0 PL=0
MOVL C00847 V=800.0 PL=0
MOVL C00848 V=800.0 PL=0
MOVL C00849 V=800.0 PL=0
MOVL C00850 V=800.0 PL=0
MOVL C00851 V=800.0 PL=0
MOVL C00852 V=800.0 PL=0
MOVL C00853 V=800.0 PL=0
MOVL C00854 V=800.0 PL=0
MOVL C00855 V=800.0 PL=0
MOVL C00856 V=800.0 PL=0
MOVL C00857 V=800.0 PL=0
MOVL C00858 V=800.0 PL=0
MOVL C00859 V=800.0 PL=0
MOVL C00860 V=800.0 PL=0
MOVL C00861 V=800.0 PL=0
MOVL C00862 V=800.0 PL=0
MOVL C00863 V=800.0 PL=0
MOVL C00864 V=800.0 PL=0
MOVL C00865 V=800.0 PL=0
MOVL C00866 V=800.0 PL=0
MOVL C00867 V=800.0 PL=0
MOVL C00868 V=800.0 PL=0
MOVL C00869 V=800.0 PL=0
MOVL C00870 V=800.0 PL=0
MOVL C00871 V=800.0 PL=0
MOVL C00872 V=800.0 PL=0
MOVL C00873 V=800.0 PL=0
MOVL C00874 V=800.0 PL=0
MOVL C00875 V=800.0 PL=0
MOVL C00876 V=800.0 PL=0
MOVL C00877 V=800.0 PL=0
MOVL C00878 V=800.0 PL=0
MOVL C00879 V=800.0 PL=0
MOVL C00880 V=800.0 PL=0
MOVL C00881 V=800.0 PL=0
MOVL C00882 V=800.0 PL=0
MOVL C00883 V=800.0 PL=0
MOVL C00884 V=800.0 PL=0
MOVL C00885 V=800.0 PL=0
MOVL C00886 V=800.0 PL=0
MOVL C00887 V=800.0 PL=0
MOVL C00888 V=800.0 PL=0
MOVL C00889 V=800.0 PL=0
MOVL C00890 V=800.0 PL=0
MOVL C00891 V=800.0 PL=0
MOVL C00892 V=800.0 PL=0
MOVL C00893 V=800.0 PL=0
MOVL C00894 V=800.0 PL=0
MOVL C00895 V=800.0 PL=0
MOVL C00896 V=800.0 PL=0
MOVL C00897 V=800.0 PL=0
MOVL C00898 V=800.0 PL=0
MOVL C00899 V=800.0 PL=0
MOVL C00900 V=800.0 PL=0
MOVL C00901 V=800.0 PL=0
MOVL C00902 V=800.0 PL=0
MOVL C00903 V=800.0 PL=0
MOVL C00904 V=800.0 PL=0
MOVL C00905 V=800.0 PL=0
MOVL C00906 V=800.0 PL=0
MOVL C00907 V=800.0 PL=0
MOVL C00908 V=800.0 PL=0
MOVL C00909 V=800.0 PL=0
MOVL C00910 V=800.0 PL=0
MOVL C00911 V=800.0 PL=0
MOVL C00912 V=800.0 PL=0
MOVL C00913 V=800.0 PL=0
MOVL C00914 V=800.0 PL=0
MOVL C00915 V=800.0 PL=0
MOVL C00916 V=800.0 PL=0
MOVL C00917 V=800.0 PL=0
MOVL C00918 V=800.0 PL=0
MOVL C00919 V=800.0 PL=0
MOVL C00920 V=800.0 PL=0
MOVL C00921 V=800.0 PL=0
MOVL C00922 V=800.0 PL=0
MOVL C00923 V=800.0 PL=0
MOVL C00924 V=800.0 PL=0
MOVL C00925 V=800.0 PL=0
MOVL C00926 V=800.0 PL=0
MOVL C00927 V=800.0 PL=0
MOVL C00928 V=800.0 PL=0
MOVL C00929 V=800.0 PL=0
MOVL C00930 V=800.0 PL=0
MOVL C00931 V=800.0 PL=0
MOVL C00932 V=800.0 PL=0
MOVL C00933 V=800.0 PL=0
MOVL C00934 V=800.0 PL=0
MOVL C00935 V=800.0 PL=0
MOVL C00936 V=800.0 PL=0
MOVL C00937 V=800.0 PL=0
MOVL C00938 V=800.0 PL=0
MOVL C00939 V=800.0 PL=0
MOVL C00940 V=800.0 PL=0
MOVL C00941 V=800.0 PL=0
MOVL C00942 V=800.0 PL=0
MOVL C00943 V=800.0 PL=0
MOVL C00944 V=800.0 PL=0
MOVL C00945 V=800.0 PL=0
MOVL C00946 V=800.0 PL=0
MOVL C00947 V=800.0 PL=0
MOVL C00948 V=800.0 PL=0
MOVL C00949 V=800.0 PL=0
MOVL C00950 V=800.0 PL=0
MOVL C00951 V=800.0 PL=0
MOVL C00952 V=800.0 PL=0
MOVL C00953 V=800.0 PL=0
MOVL C00954 V=800.0 PL=0
MOVL C00955 V=800.0 PL=0
MOVL C00956 V=800.0 PL=0
MOVL C00957 V=800.0 PL=0
MOVL C00958 V=800.0 PL=0
MOVL C00959 V=800.0 PL=0
MOVL C00960 V=800.0 PL=0
MOVL C00961 V=800.0 PL=0
MOVL C00962 V=800.0 PL=0
MOVL C00963 V=800.0 PL=0
MOVL C00964 V=800.0 PL=0
MOVL C00965 V=800.0 PL=0
MOVL C00966 V=800.0 PL=0
MOVL C00967 V=800.0 PL=0
MOVL C00968 V=800.0 PL=0
MOVL C00969 V=800.0 PL=0
MOVL C00970 V=800.0 PL=0
MOVL C00971 V=800.0 PL=0
MOVL C00972 V=800.0 PL=0
MOVL C00973 V=800.0 PL=0
MOVL C00974 V=800.0 PL=0
MOVL C00975 V=800.0 PL=0
MOVL C00976 V=800.0 PL=0
MOVL C00977 V=800.0 PL=0
MOVL C00978 V=800.0 PL=0
MOVL C00979 V=800.0 PL=0
MOVL C00980 V=800.0 PL=0
MOVL C00981 V=800.0 PL=0
MOVL C00982 V=800.0 PL=0
MOVL C00983 V=800.0 PL=0
MOVL C00984 V=800.0 PL=0
MOVL C00985 V=800.0 PL=0
MOVL C00986 V=800.0 PL=0
MOVL C00987 V=800.0 PL=0
MOVL C00988 V=800.0 PL=0
MOVL C00989 V=800.0 PL=0
MOVL C00990 V=800.0 PL=0
MOVL C00991 V=800.0 PL=0
MOVL C00992 V=800.0 PL=0
MOVL C00993 V=800.0 PL=0
MOVL C00994 V=800.0 PL=0
MOVL C00995 V=800.0 PL=0
MOVL C00996 V=800.0 PL=0
MOVL C00997 V=800.0 PL=0
MOVL C00998 V=800.0 PL=0
MOVL C00999 V=800.0 PL=0
MOVL C01000 V=800.0 PL=0
MOVL C01001 V=800.0 PL=0
MOVL C01002 V=800.0 PL=0
MOVL C01003 V=800.0 PL=0
MOVL C01004 V=800.0 PL=0
MOVL C01005 V=800.0 PL=0
MOVL C01006 V=800.0 PL=0
MOVL C01007 V=800.0 PL=0
MOVL C01008 V=800.0 PL=0
MOVL C01009 V=800.0 PL=0
MOVL C01010 V=800.0 PL=0
MOVL C01011 V=800.0 PL=0
MOVL C01012 V=800.0 PL=0
MOVL C01013 V=800.0 PL=0
MOVL C01014 V=800.0 PL=0
MOVL C01015 V=800.0 PL=0
MOVL C01016 V=800.0 PL=0
MOVL C01017 V=800.0 PL=0
MOVL C01018 V=800.0 PL=0
MOVL C01019 V=800.0 PL=0
MOVL C01020 V=800.0 PL=0
MOVL C01021 V=800.0 PL=0
MOVL C01022 V=800.0 PL=0
MOVL C01023 V=800.0 PL=0
MOVL C01024 V=800.0 PL=0
MOVL C01025 V=800.0 PL=0
MOVL C01026 V=800.0 PL=0
MOVL C01027 V=800.0 PL=0
MOVL C01028 V=800.0 PL=0
MOVL C01029 V=800.0 PL=0
MOVL C01030 V=800.0 PL=0
MOVL C01031 V=800.0 PL=0
MOVL C01032 V=800.0 PL=0
MOVL C01033 V=800.0 PL=0
MOVL C01034 V=800.0 PL=0
MOVL C01035 V=800.0 PL=0
MOVL C01036 V=800.0 PL=0
MOVL C01037 V=800.0 PL=0
MOVL C01038 V=800.0 PL=0
MOVL C01039 V=800.0 PL=0
MOVL C01040 V=800.0 PL=0
MOVL C01041 V=800.0 PL=0
MOVL C01042 V=800.0 PL=0
MOVL C01043 V=800.0 PL=0
MOVL C01044 V=800.0 PL=0
MOVL C01045 V=800.0 PL=0
MOVL C01046 V=800.0 PL=0
MOVL C01047 V=800.0 PL=0
MOVL C01048 V=800.0 PL=0
MOVL C01049 V=800.0 PL=0
MOVL C01050 V=800.0 PL=0
MOVL C01051 V=800.0 PL=0
MOVL C01052 V=800.0 PL=0
MOVL C01053 V=800.0 PL=0
MOVL C01054 V=800.0 PL=0
MOVL C01055 V=800.0 PL=0
MOVL C01056 V=800.0 PL=0
MOVL C01057 V=800.0 PL=0
MOVL C01058 V=800.0 PL=0
MOVL C01059 V=800.0 PL=0
MOVL C01060 V=800.0 PL=0
MOVL C01061 V=800.0 PL=0
MOVL C01062 V=800.0 PL=0
MOVL C01063 V=800.0 PL=0
MOVL C01064 V=800.0 PL=0
MOVL C01065 V=800.0 PL=0
MOVL C01066 V=800.0 PL=0
MOVL C01067 V=800.0 PL=0
MOVL C01068 V=800.0 PL=0
MOVL C01069 V=800.0 PL=0
MOVL C01070 V=800.0 PL=0
MOVL C01071 V=800.0 PL=0
MOVL C01072 V=800.0 PL=0
MOVL C01073 V=800.0 PL=0
MOVL C01074 V=800.0 PL=0
MOVL C01075 V=800.0 PL=0
MOVL C01076 V=800.0 PL=0
MOVL C01077 V=800.0 PL=0
MOVL C01078 V=800.0 PL=0
MOVL C01079 V=800.0 PL=0
MOVL C01080 V=800.0 PL=0
MOVL C01081 V=800.0 PL=0
MOVL C01082 V=800.0 PL=0
MOVL C01083 V=800.0 PL=0
MOVL C01084 V=800.0 PL=0
MOVL C01085 V=800.0 PL=0
MOVL C01086 V=800.0 PL=0
MOVL C01087 V=800.0 PL=0
MOVL C01088 V=800.0 PL=0
MOVL C01089 V=800.0 PL=0
MOVL C01090 V=800.0 PL=0
MOVL C01091 V=800.0 PL=0
MOVL C01092 V=800.0 PL=0
MOVL C01093 V=800.0 PL=0
MOVL C01094 V=800.0 PL=0
MOVL C01095 V=800.0 PL=0
MOVL C01096 V=800.0 PL=0
MOVL C01097 V=800.0 PL=0
MOVL C01098 V=800.0 PL=0
MOVL C01099 V=800.0 PL=0
MOVL C01100 V=800.0 PL=0
MOVL C01101 V=800.0 PL=0
MOVL C01102 V=800.0 PL=0
MOVL C01103 V=800.0 PL=0
MOVL C01104 V=800.0 PL=0
MOVL C01105 V=800.0 PL=0
MOVL C01106 V=800.0 PL=0
MOVL C01107 V=800.0 PL=0
MOVL C01108 V=800.0 PL=0
MOVL C01109 V=800.0 PL=0
MOVL C01110 V=800.0 PL=0
MOVL C01111 V=800.0 PL=0
MOVL C01112 V=800.0 PL=0
MOVL C01113 V=800.0 PL=0
MOVL C01114 V=800.0 PL=0
MOVL C01115 V=800.0 PL=0
MOVL C01116 V=800.0 PL=0
MOVL C01117 V=800.0 PL=0
MOVL C01118 V=800.0 PL=0
MOVL C01119 V=800.0 PL=0
MOVL C01120 V=800.0 PL=0
MOVL C01121 V=800.0 PL=0
MOVL C01122 V=800.0 PL=0
MOVL C01123 V=800.0 PL=0
MOVL C01124 V=800.0 PL=0
MOVL C01125 V=800.0 PL=0
MOVL C01126 V=800.0 PL=0
MOVL C01127 V=800.0 PL=0
MOVL C01128 V=800.0 PL=0
MOVL C01129 V=800.0 PL=0
MOVL C01130 V=800.0 PL=0
MOVL C01131 V=800.0 PL=0
MOVL C01132 V=800.0 PL=0
MOVL C01133 V=800.0 PL=0
MOVL C01134 V=800.0 PL=0
MOVL C01135 V=800.0 PL=0
MOVL C01136 V=800.0 PL=0
MOVL C01137 V=800.0 PL=0
MOVL C01138 V=800.0 PL=0
MOVL C01139 V=800.0 PL=0
MOVL C01140 V=800.0 PL=0
MOVL C01141 V=800.0 PL=0
MOVL C01142 V=800.0 PL=0
MOVL C01143 V=800.0 PL=0
MOVL C01144 V=800.0 PL=0
MOVL C01145 V=800.0 PL=0
MOVL C01146 V=800.0 PL=0
MOVL C01147 V=800.0 PL=0
MOVL C01148 V=800.0 PL=0
MOVL C01149 V=800.0 PL=0
MOVL C01150 V=800.0 PL=0
MOVL C01151 V=800.0 PL=0
MOVL C01152 V=800.0 PL=0
MOVL C01153 V=800.0 PL=0
MOVL C01154 V=800.0 PL=0
MOVL C01155 V=800.0 PL=0
MOVL C01156 V=800.0 PL=0
MOVL C01157 V=800.0 PL=0
MOVL C01158 V=800.0 PL=0
MOVL C01159 V=800.0 PL=0
MOVL C01160 V=800.0 PL=0
MOVL C01161 V=800.0 PL=0
MOVL C01162 V=800.0 PL=0
MOVL C01163 V=800.0 PL=0
MOVL C01164 V=800.0 PL=0
MOVL C01165 V=800.0 PL=0
MOVL C01166 V=800.0 PL=0
MOVL C01167 V=800.0 PL=0
MOVL C01168 V=800.0 PL=0
MOVL C01169 V=800.0 PL=0
MOVL C01170 V=800.0 PL=0
MOVL C01171 V=800.0 PL=0
MOVL C01172 V=800.0 PL=0
MOVL C01173 V=800.0 PL=0
MOVL C01174 V=800.0 PL=0
MOVL C01175 V=800.0 PL=0
MOVL C01176 V=800.0 PL=0
MOVL C01177 V=800.0 PL=0
MOVL C01178 V=800.0 PL=0
MOVL C01179 V=800.0 PL=0
MOVL C01180 V=800.0 PL=0
MOVL C01181 V=800.0 PL=0
MOVL C01182 V=800.0 PL=0
MOVL C01183 V=800.0 PL=0
MOVL C01184 V=800.0 PL=0
MOVL C01185 V=800.0 PL=0
MOVL C01186 V=800.0 PL=0
MOVL C01187 V=800.0 PL=0
MOVL C01188 V=800.0 PL=0
MOVL C01189 V=800.0 PL=0
MOVL C01190 V=800.0 PL=0
MOVL C01191 V=800.0 PL=0
MOVL C01192 V=800.0 PL=0
MOVL C01193 V=800.0 PL=0
MOVL C01194 V=800.0 PL=0
MOVL C01195 V=800.0 PL=0
MOVL C01196 V=800.0 PL=0
MOVL C01197 V=800.0 PL=0
MOVL C01198 V=800.0 PL=0
MOVL C01199 V=800.0 PL=0
MOVL C01200 V=800.0 PL=0
MOVL C01201 V=800.0 PL=0
MOVL C01202 V=800.0 PL=0
MOVL C01203 V=800.0 PL=0
MOVL C01204 V=800.0 PL=0
MOVL C01205 V=800.0 PL=0
MOVL C01206 V=800.0 PL=0
MOVL C01207 V=800.0 PL=0
MOVL C01208 V=800.0 PL=0
MOVL C01209 V=800.0 PL=0
MOVL C01210 V=800.0 PL=0
MOVL C01211 V=800.0 PL=0
MOVL C01212 V=800.0 PL=0
MOVL C01213 V=800.0 PL=0
MOVL C01214 V=800.0 PL=0
MOVL C01215 V=800.0 PL=0
MOVL C01216 V=800.0 PL=0
MOVL C01217 V=800.0 PL=0
MOVL C01218 V=800.0 PL=0
MOVL C01219 V=800.0 PL=0
MOVL C01220 V=800.0 PL=0
MOVL C01221 V=800.0 PL=0
MOVL C01222 V=800.0 PL=0
MOVL C01223 V=800.0 PL=0
MOVL C01224 V=800.0 PL=0
MOVL C01225 V=800.0 PL=0
MOVL C01226 V=800.0 PL=0
MOVL C01227 V=800.0 PL=0
MOVL C01228 V=800.0 PL=0
MOVL C01229 V=800.0 PL=0
MOVL C01230 V=800.0 PL=0
MOVL C01231 V=800.0 PL=0
MOVL C01232 V=800.0 PL=0
MOVL C01233 V=800.0 PL=0
MOVL C01234 V=800.0 PL=0
MOVL C01235 V=800.0 PL=0
MOVL C01236 V=800.0 PL=0
MOVL C01237 V=800.0 PL=0
MOVL C01238 V=800.0 PL=0
MOVL C01239 V=800.0 PL=0
MOVL C01240 V=800.0 PL=0
MOVL C01241 V=800.0 PL=0
MOVL C01242 V=800.0 PL=0
MOVL C01243 V=800.0 PL=0
MOVL C01244 V=800.0 PL=0
MOVL C01245 V=800.0 PL=0
MOVL C01246 V=800.0 PL=0
MOVL C01247 V=800.0 PL=0
MOVL C01248 V=800.0 PL=0
MOVL C01249 V=800.0 PL=0
MOVL C01250 V=800.0 PL=0
MOVL C01251 V=800.0 PL=0
MOVL C01252 V=800.0 PL=0
MOVL C01253 V=800.0 PL=0
MOVL C01254 V=800.0 PL=0
MOVL C01255 V=800.0 PL=0
MOVL C01256 V=800.0 PL=0
MOVL C01257 V=800.0 PL=0
MOVL C01258 V=800.0 PL=0
MOVL C01259 V=800.0 PL=0
MOVL C01260 V=800.0 PL=0
MOVL C01261 V=800.0 PL=0
MOVL C01262 V=800.0 PL=0
MOVL C01263 V=800.0 PL=0
MOVL C01264 V=800.0 PL=0
MOVL C01265 V=800.0 PL=0
MOVL C01266 V=800.0 PL=0
MOVL C01267 V=800.0 PL=0
MOVL C01268 V=800.0 PL=0
MOVL C01269 V=800.0 PL=0
MOVL C01270 V=800.0 PL=0
MOVL C01271 V=800.0 PL=0
MOVL C01272 V=800.0 PL=0
MOVL C01273 V=800.0 PL=0
MOVL C01274 V=800.0 PL=0
MOVL C01275 V=800.0 PL=0
MOVL C01276 V=800.0 PL=0
MOVL C01277 V=800.0 PL=0
MOVL C01278 V=800.0 PL=0
MOVL C01279 V=800.0 PL=0
MOVL C01280 V=800.0 PL=0
MOVL C01281 V=800.0 PL=0
MOVL C01282 V=800.0 PL=0
MOVL C01283 V=800.0 PL=0
MOVL C01284 V=800.0 PL=0
MOVL C01285 V=800.0 PL=0
MOVL C01286 V=800.0 PL=0
MOVL C01287 V=800.0 PL=0
MOVL C01288 V=800.0 PL=0
MOVL C01289 V=800.0 PL=0
MOVL C01290 V=800.0 PL=0
MOVL C01291 V=800.0 PL=0
MOVL C01292 V=800.0 PL=0
MOVL C01293 V=800.0 PL=0
MOVL C01294 V=800.0 PL=0
MOVL C01295 V=800.0 PL=0
MOVL C01296 V=800.0 PL=0
MOVL C01297 V=800.0 PL=0
MOVL C01298 V=800.0 PL=0
MOVL C01299 V=800.0 PL=0
MOVL C01300 V=800.0 PL=0
MOVL C01301 V=800.0 PL=0
MOVL C01302 V=800.0 PL=0
MOVL C01303 V=800.0 PL=0
MOVL C01304 V=800.0 PL=0
MOVL C01305 V=800.0 PL=0
MOVL C01306 V=800.0 PL=0
MOVL C01307 V=800.0 PL=0
MOVL C01308 V=800.0 PL=0
MOVL C01309 V=800.0 PL=0
MOVL C01310 V=800.0 PL=0
MOVL C01311 V=800.0 PL=0
MOVL C01312 V=800.0 PL=0
MOVL C01313 V=800.0 PL=0
MOVL C01314 V=800.0 PL=0
MOVL C01315 V=800.0 PL=0
MOVL C01316 V=800.0 PL=0
MOVL C01317 V=800.0 PL=0
MOVL C01318 V=800.0 PL=0
MOVL C01319 V=800.0 PL=0
MOVL C01320 V=800.0 PL=0
MOVL C01321 V=800.0 PL=0
MOVL C01322 V=800.0 PL=0
MOVL C01323 V=800.0 PL=0
MOVL C01324 V=800.0 PL=0
MOVL C01325 V=800.0 PL=0
MOVL C01326 V=800.0 PL=0
MOVL C01327 V=800.0 PL=0
MOVL C01328 V=800.0 PL=0
MOVL C01329 V=800.0 PL=0
MOVL C01330 V=800.0 PL=0
MOVL C01331 V=800.0 PL=0
MOVL C01332 V=800.0 PL=0
MOVL C01333 V=800.0 PL=0
MOVL C01334 V=800.0 PL=0
MOVL C01335 V=800.0 PL=0
MOVL C01336 V=800.0 PL=0
MOVL C01337 V=800.0 PL=0
MOVL C01338 V=800.0 PL=0
MOVL C01339 V=800.0 PL=0
MOVL C01340 V=800.0 PL=0
MOVL C01341 V=800.0 PL=0
MOVL C01342 V=800.0 PL=0
MOVL C01343 V=800.0 PL=0
MOVL C01344 V=800.0 PL=0
MOVL C01345 V=800.0 PL=0
MOVL C01346 V=800.0 PL=0
MOVL C01347 V=800.0 PL=0
MOVL C01348 V=800.0 PL=0
MOVL C01349 V=800.0 PL=0
MOVL C01350 V=800.0 PL=0
MOVL C01351 V=800.0 PL=0
MOVL C01352 V=800.0 PL=0
MOVL C01353 V=800.0 PL=0
MOVL C01354 V=800.0 PL=0
MOVL C01355 V=800.0 PL=0
MOVL C01356 V=800.0 PL=0
MOVL C01357 V=800.0 PL=0
MOVL C01358 V=800.0 PL=0
MOVL C01359 V=800.0 PL=0
MOVL C01360 V=800.0 PL=0
MOVL C01361 V=800.0 PL=0
MOVL C01362 V=800.0 PL=0
MOVL C01363 V=800.0 PL=0
MOVL C01364 V=800.0 PL=0
MOVL C01365 V=800.0 PL=0
MOVL C01366 V=800.0 PL=0
MOVL C01367 V=800.0 PL=0
MOVL C01368 V=800.0 PL=0
MOVL C01369 V=800.0 PL=0
MOVL C01370 V=800.0 PL=0
MOVL C01371 V=800.0 PL=0
MOVL C01372 V=800.0 PL=0
MOVL C01373 V=800.0 PL=0
MOVL C01374 V=800.0 PL=0
MOVL C01375 V=800.0 PL=0
MOVL C01376 V=800.0 PL=0
MOVL C01377 V=800.0 PL=0
MOVL C01378 V=800.0 PL=0
MOVL C01379 V=800.0 PL=0
MOVL C01380 V=800.0 PL=0
MOVL C01381 V=800.0 PL=0
MOVL C01382 V=800.0 PL=0
MOVL C01383 V=800.0 PL=0
MOVL C01384 V=800.0 PL=0
MOVL C01385 V=800.0 PL=0
MOVL C01386 V=800.0 PL=0
MOVL C01387 V=800.0 PL=0
MOVL C01388 V=800.0 PL=0
MOVL C01389 V=800.0 PL=0
MOVL C01390 V=800.0 PL=0
MOVL C01391 V=800.0 PL=0
MOVL C01392 V=800.0 PL=0
MOVL C01393 V=800.0 PL=0
MOVL C01394 V=800.0 PL=0
MOVL C01395 V=800.0 PL=0
MOVL C01396 V=800.0 PL=0
MOVL C01397 V=800.0 PL=0
MOVL C01398 V=800.0 PL=0
MOVL C01399 V=800.0 PL=0
MOVL C01400 V=800.0 PL=0
MOVL C01401 V=800.0 PL=0
MOVL C01402 V=800.0 PL=0
MOVL C01403 V=800.0 PL=0
MOVL C01404 V=800.0 PL=0
MOVL C01405 V=800.0 PL=0
MOVL C01406 V=800.0 PL=0
MOVL C01407 V=800.0 PL=0
MOVL C01408 V=800.0 PL=0
MOVL C01409 V=800.0 PL=0
MOVL C01410 V=800.0 PL=0
MOVL C01411 V=800.0 PL=0
MOVL C01412 V=800.0 PL=0
MOVL C01413 V=800.0 PL=0
MOVL C01414 V=800.0 PL=0
MOVL C01415 V=800.0 PL=0
MOVL C01416 V=800.0 PL=0
MOVL C01417 V=800.0 PL=0
MOVL C01418 V=800.0 PL=0
MOVL C01419 V=800.0 PL=0
MOVL C01420 V=800.0 PL=0
MOVL C01421 V=800.0 PL=0
MOVL C01422 V=800.0 PL=0
MOVL C01423 V=800.0 PL=0
MOVL C01424 V=800.0 PL=0
MOVL C01425 V=800.0 PL=0
MOVL C01426 V=800.0 PL=0
MOVL C01427 V=800.0 PL=0
MOVL C01428 V=800.0 PL=0
MOVL C01429 V=800.0 PL=0
MOVL C01430 V=800.0 PL=0
MOVL C01431 V=800.0 PL=0
MOVL C01432 V=800.0 PL=0
MOVL C01433 V=800.0 PL=0
MOVL C01434 V=800.0 PL=0
MOVL C01435 V=800.0 PL=0
MOVL C01436 V=800.0 PL=0
MOVL C01437 V=800.0 PL=0
MOVL C01438 V=800.0 PL=0
MOVL C01439 V=800.0 PL=0
MOVL C01440 V=800.0 PL=0
MOVL C01441 V=800.0 PL=0
MOVL C01442 V=800.0 PL=0
MOVL C01443 V=800.0 PL=0
MOVL C01444 V=800.0 PL=0
MOVL C01445 V=800.0 PL=0
MOVL C01446 V=800.0 PL=0
MOVL C01447 V=800.0 PL=0
MOVL C01448 V=800.0 PL=0
MOVL C01449 V=800.0 PL=0
MOVL C01450 V=800.0 PL=0
MOVL C01451 V=800.0 PL=0
MOVL C01452 V=800.0 PL=0
MOVL C01453 V=800.0 PL=0
MOVL C01454 V=800.0 PL=0
MOVL C01455 V=800.0 PL=0
MOVL C01456 V=800.0 PL=0
MOVL C01457 V=800.0 PL=0
MOVL C01458 V=800.0 PL=0
MOVL C01459 V=800.0 PL=0
MOVL C01460 V=800.0 PL=0
MOVL C01461 V=800.0 PL=0
MOVL C01462 V=800.0 PL=0
MOVL C01463 V=800.0 PL=0
MOVL C01464 V=800.0 PL=0
MOVL C01465 V=800.0 PL=0
MOVL C01466 V=800.0 PL=0
MOVL C01467 V=800.0 PL=0
MOVL C01468 V=800.0 PL=0
MOVL C01469 V=800.0 PL=0
MOVL C01470 V=800.0 PL=0
MOVL C01471 V=800.0 PL=0
MOVL C01472 V=800.0 PL=0
MOVL C01473 V=800.0 PL=0
MOVL C01474 V=800.0 PL=0
MOVL C01475 V=800.0 PL=0
MOVL C01476 V=800.0 PL=0
MOVL C01477 V=800.0 PL=0
MOVL C01478 V=800.0 PL=0
MOVL C01479 V=800.0 PL=0
MOVL C01480 V=800.0 PL=0
MOVL C01481 V=800.0 PL=0
MOVL C01482 V=800.0 PL=0
MOVL C01483 V=800.0 PL=0
MOVL C01484 V=800.0 PL=0
MOVL C01485 V=800.0 PL=0
MOVL C01486 V=800.0 PL=0
MOVL C01487 V=800.0 PL=0
MOVL C01488 V=800.0 PL=0
MOVL C01489 V=800.0 PL=0
MOVL C01490 V=800.0 PL=0
MOVL C01491 V=800.0 PL=0
MOVL C01492 V=800.0 PL=0
MOVL C01493 V=800.0 PL=0
MOVL C01494 V=800.0 PL=0
MOVL C01495 V=800.0 PL=0
MOVL C01496 V=800.0 PL=0
MOVL C01497 V=800.0 PL=0
MOVL C01498 V=800.0 PL=0
MOVL C01499 V=800.0 PL=0
MOVL C01500 V=800.0 PL=0
MOVL C01501 V=800.0 PL=0
MOVL C01502 V=800.0 PL=0
MOVL C01503 V=800.0 PL=0
MOVL C01504 V=800.0 PL=0
MOVL C01505 V=800.0 PL=0
MOVL C01506 V=800.0 PL=0
MOVL C01507 V=800.0 PL=0
MOVL C01508 V=800.0 PL=0
MOVL C01509 V=800.0 PL=0
MOVL C01510 V=800.0 PL=0
MOVL C01511 V=800.0 PL=0
MOVL C01512 V=800.0 PL=0
MOVL C01513 V=800.0 PL=0
MOVL C01514 V=800.0 PL=0
MOVL C01515 V=800.0 PL=0
MOVL C01516 V=800.0 PL=0
MOVL C01517 V=800.0 PL=0
MOVL C01518 V=800.0 PL=0
MOVL C01519 V=800.0 PL=0
MOVL C01520 V=800.0 PL=0
MOVL C01521 V=800.0 PL=0
MOVL C01522 V=800.0 PL=0
MOVL C01523 V=800.0 PL=0
MOVL C01524 V=800.0 PL=0
MOVL C01525 V=800.0 PL=0
MOVL C01526 V=800.0 PL=0
MOVL C01527 V=800.0 PL=0
MOVL C01528 V=800.0 PL=0
MOVL C01529 V=800.0 PL=0
MOVL C01530 V=800.0 PL=0
MOVL C01531 V=800.0 PL=0
MOVL C01532 V=800.0 PL=0
MOVL C01533 V=800.0 PL=0
MOVL C01534 V=800.0 PL=0
MOVL C01535 V=800.0 PL=0
MOVL C01536 V=800.0 PL=0
MOVL C01537 V=800.0 PL=0
MOVL C01538 V=800.0 PL=0
MOVL C01539 V=800.0 PL=0
MOVL C01540 V=800.0 PL=0
MOVL C01541 V=800.0 PL=0
MOVL C01542 V=800.0 PL=0
MOVL C01543 V=800.0 PL=0
MOVL C01544 V=800.0 PL=0
MOVL C01545 V=800.0 PL=0
MOVL C01546 V=800.0 PL=0
MOVL C01547 V=800.0 PL=0
MOVL C01548 V=800.0 PL=0
MOVL C01549 V=800.0 PL=0
MOVL C01550 V=800.0 PL=0
MOVL C01551 V=800.0 PL=0
MOVL C01552 V=800.0 PL=0
MOVL C01553 V=800.0 PL=0
MOVL C01554 V=800.0 PL=0
MOVL C01555 V=800.0 PL=0
MOVL C01556 V=800.0 PL=0
MOVL C01557 V=800.0 PL=0
MOVL C01558 V=800.0 PL=0
MOVL C01559 V=800.0 PL=0
MOVL C01560 V=800.0 PL=0
MOVL C01561 V=800.0 PL=0
MOVL C01562 V=800.0 PL=0
MOVL C01563 V=800.0 PL=0
MOVL C01564 V=800.0 PL=0
MOVL C01565 V=800.0 PL=0
MOVL C01566 V=800.0 PL=0
MOVL C01567 V=800.0 PL=0
MOVL C01568 V=800.0 PL=0
MOVL C01569 V=800.0 PL=0
MOVL C01570 V=800.0 PL=0
MOVL C01571 V=800.0 PL=0
MOVL C01572 V=800.0 PL=0
MOVL C01573 V=800.0 PL=0
MOVL C01574 V=800.0 PL=0
MOVL C01575 V=800.0 PL=0
MOVL C01576 V=800.0 PL=0
MOVL C01577 V=800.0 PL=0
MOVL C01578 V=800.0 PL=0
MOVL C01579 V=800.0 PL=0
MOVL C01580 V=800.0 PL=0
MOVL C01581 V=800.0 PL=0
MOVL C01582 V=800.0 PL=0
MOVL C01583 V=800.0 PL=0
MOVL C01584 V=800.0 PL=0
MOVL C01585 V=800.0 PL=0
MOVL C01586 V=800.0 PL=0
MOVL C01587 V=800.0 PL=0
MOVL C01588 V=800.0 PL=0
MOVL C01589 V=800.0 PL=0
MOVL C01590 V=800.0 PL=0
MOVL C01591 V=800.0 PL=0
MOVL C01592 V=800.0 PL=0
MOVL C01593 V=800.0 PL=0
MOVL C01594 V=800.0 PL=0
MOVL C01595 V=800.0 PL=0
MOVL C01596 V=800.0 PL=0
MOVL C01597 V=800.0 PL=0
MOVL C01598 V=800.0 PL=0
MOVL C01599 V=800.0 PL=0
MOVL C01600 V=800.0 PL=0
MOVL C01601 V=800.0 PL=0
MOVL C01602 V=800.0 PL=0
MOVL C01603 V=800.0 PL=0
MOVL C01604 V=800.0 PL=0
MOVL C01605 V=800.0 PL=0
MOVL C01606 V=800.0 PL=0
MOVL C01607 V=800.0 PL=0
MOVL C01608 V=800.0 PL=0
MOVL C01609 V=800.0 PL=0
MOVL C01610 V=800.0 PL=0
MOVL C01611 V=800.0 PL=0
MOVL C01612 V=800.0 PL=0
MOVL C01613 V=800.0 PL=0
MOVL C01614 V=800.0 PL=0
MOVL C01615 V=800.0 PL=0
MOVL C01616 V=800.0 PL=0
MOVL C01617 V=800.0 PL=0
MOVL C01618 V=800.0 PL=0
MOVL C01619 V=800.0 PL=0
MOVL C01620 V=800.0 PL=0
MOVL C01621 V=800.0 PL=0
MOVL C01622 V=800.0 PL=0
MOVL C01623 V=800.0 PL=0
MOVL C01624 V=800.0 PL=0
MOVL C01625 V=800.0 PL=0
MOVL C01626 V=800.0 PL=0
MOVL C01627 V=800.0 PL=0
MOVL C01628 V=800.0 PL=0
MOVL C01629 V=800.0 PL=0
MOVL C01630 V=800.0 PL=0
MOVL C01631 V=800.0 PL=0
MOVL C01632 V=800.0 PL=0
MOVL C01633 V=800.0 PL=0
MOVL C01634 V=800.0 PL=0
MOVL C01635 V=800.0 PL=0
MOVL C01636 V=800.0 PL=0
MOVL C01637 V=800.0 PL=0
MOVL C01638 V=800.0 PL=0
MOVL C01639 V=800.0 PL=0
MOVL C01640 V=800.0 PL=0
MOVL C01641 V=800.0 PL=0
MOVL C01642 V=800.0 PL=0
MOVL C01643 V=800.0 PL=0
MOVL C01644 V=800.0 PL=0
MOVL C01645 V=800.0 PL=0
MOVL C01646 V=800.0 PL=0
MOVL C01647 V=800.0 PL=0
MOVL C01648 V=800.0 PL=0
MOVL C01649 V=800.0 PL=0
MOVL C01650 V=800.0 PL=0
MOVL C01651 V=800.0 PL=0
MOVL C01652 V=800.0 PL=0
MOVL C01653 V=800.0 PL=0
MOVL C01654 V=800.0 PL=0
MOVL C01655 V=800.0 PL=0
MOVL C01656 V=800.0 PL=0
MOVL C01657 V=800.0 PL=0
MOVL C01658 V=800.0 PL=0
MOVL C01659 V=800.0 PL=0
MOVL C01660 V=800.0 PL=0
MOVL C01661 V=800.0 PL=0
MOVL C01662 V=800.0 PL=0
MOVL C01663 V=800.0 PL=0
MOVL C01664 V=800.0 PL=0
MOVL C01665 V=800.0 PL=0
MOVL C01666 V=800.0 PL=0
MOVL C01667 V=800.0 PL=0
MOVL C01668 V=800.0 PL=0
MOVL C01669 V=800.0 PL=0
MOVL C01670 V=800.0 PL=0
MOVL C01671 V=800.0 PL=0
MOVL C01672 V=800.0 PL=0
MOVL C01673 V=800.0 PL=0
MOVL C01674 V=800.0 PL=0
MOVL C01675 V=800.0 PL=0
MOVL C01676 V=800.0 PL=0
MOVL C01677 V=800.0 PL=0
MOVL C01678 V=800.0 PL=0
MOVL C01679 V=800.0 PL=0
MOVL C01680 V=800.0 PL=0
MOVL C01681 V=800.0 PL=0
MOVL C01682 V=800.0 PL=0
MOVL C01683 V=800.0 PL=0
MOVL C01684 V=800.0 PL=0
MOVL C01685 V=800.0 PL=0
MOVL C01686 V=800.0 PL=0
MOVL C01687 V=800.0 PL=0
MOVL C01688 V=800.0 PL=0
MOVL C01689 V=800.0 PL=0
MOVL C01690 V=800.0 PL=0
MOVL C01691 V=800.0 PL=0
MOVL C01692 V=800.0 PL=0
MOVL C01693 V=800.0 PL=0
MOVL C01694 V=800.0 PL=0
MOVL C01695 V=800.0 PL=0
MOVL C01696 V=800.0 PL=0
MOVL C01697 V=800.0 PL=0
MOVL C01698 V=800.0 PL=0
MOVL C01699 V=800.0 PL=0
MOVL C01700 V=800.0 PL=0
MOVL C01701 V=800.0 PL=0
MOVL C01702 V=800.0 PL=0
MOVL C01703 V=800.0 PL=0
MOVL C01704 V=800.0 PL=0
MOVL C01705 V=800.0 PL=0
MOVL C01706 V=800.0 PL=0
MOVL C01707 V=800.0 PL=0
MOVL C01708 V=800.0 PL=0
MOVL C01709 V=800.0 PL=0
MOVL C01710 V=800.0 PL=0
MOVL C01711 V=800.0 PL=0
MOVL C01712 V=800.0 PL=0
MOVL C01713 V=800.0 PL=0
MOVL C01714 V=800.0 PL=0
MOVL C01715 V=800.0 PL=0
MOVL C01716 V=800.0 PL=0
MOVL C01717 V=800.0 PL=0
MOVL C01718 V=800.0 PL=0
MOVL C01719 V=800.0 PL=0
MOVL C01720 V=800.0 PL=0
MOVL C01721 V=800.0 PL=0
MOVL C01722 V=800.0 PL=0
MOVL C01723 V=800.0 PL=0
MOVL C01724 V=800.0 PL=0
MOVL C01725 V=800.0 PL=0
MOVL C01726 V=800.0 PL=0
MOVL C01727 V=800.0 PL=0
MOVL C01728 V=800.0 PL=0
MOVL C01729 V=800.0 PL=0
MOVL C01730 V=800.0 PL=0
MOVL C01731 V=800.0 PL=0
MOVL C01732 V=800.0 PL=0
MOVL C01733 V=800.0 PL=0
MOVL C01734 V=800.0 PL=0
MOVL C01735 V=800.0 PL=0
MOVL C01736 V=800.0 PL=0
MOVL C01737 V=800.0 PL=0
MOVL C01738 V=800.0 PL=0
MOVL C01739 V=800.0 PL=0
MOVL C01740 V=800.0 PL=0
MOVL C01741 V=800.0 PL=0
MOVL C01742 V=800.0 PL=0
MOVL C01743 V=800.0 PL=0
MOVL C01744 V=800.0 PL=0
MOVL C01745 V=800.0 PL=0
MOVL C01746 V=800.0 PL=0
MOVL C01747 V=800.0 PL=0
MOVL C01748 V=800.0 PL=0
MOVL C01749 V=800.0 PL=0
MOVL C01750 V=800.0 PL=0
MOVL C01751 V=800.0 PL=0
MOVL C01752 V=800.0 PL=0
MOVL C01753 V=800.0 PL=0
MOVL C01754 V=800.0 PL=0
MOVL C01755 V=800.0 PL=0
MOVL C01756 V=800.0 PL=0
MOVL C01757 V=800.0 PL=0
MOVL C01758 V=800.0 PL=0
MOVL C01759 V=800.0 PL=0
MOVL C01760 V=800.0 PL=0
MOVL C01761 V=800.0 PL=0
MOVL C01762 V=800.0 PL=0
MOVL C01763 V=800.0 PL=0
MOVL C01764 V=800.0 PL=0
MOVL C01765 V=800.0 PL=0
MOVL C01766 V=800.0 PL=0
MOVL C01767 V=800.0 PL=0
MOVL C01768 V=800.0 PL=0
MOVL C01769 V=800.0 PL=0
MOVL C01770 V=800.0 PL=0
MOVL C01771 V=800.0 PL=0
MOVL C01772 V=800.0 PL=0
MOVL C01773 V=800.0 PL=0
MOVL C01774 V=800.0 PL=0
MOVL C01775 V=800.0 PL=0
MOVL C01776 V=800.0 PL=0
MOVL C01777 V=800.0 PL=0
MOVL C01778 V=800.0 PL=0
MOVL C01779 V=800.0 PL=0
MOVL C01780 V=800.0 PL=0
MOVL C01781 V=800.0 PL=0
MOVL C01782 V=800.0 PL=0
MOVL C01783 V=800.0 PL=0
MOVL C01784 V=800.0 PL=0
MOVL C01785 V=800.0 PL=0
MOVL C01786 V=800.0 PL=0
MOVL C01787 V=800.0 PL=0
MOVL C01788 V=800.0 PL=0
MOVL C01789 V=800.0 PL=0
MOVL C01790 V=800.0 PL=0
MOVL C01791 V=800.0 PL=0
MOVL C01792 V=800.0 PL=0
MOVL C01793 V=800.0 PL=0
MOVL C01794 V=800.0 PL=0
MOVL C01795 V=800.0 PL=0
MOVL C01796 V=800.0 PL=0
MOVL C01797 V=800.0 PL=0
MOVL C01798 V=800.0 PL=0
MOVL C01799 V=800.0 PL=0
MOVL C01800 V=800.0 PL=0
MOVL C01801 V=800.0 PL=0
MOVL C01802 V=800.0 PL=0
MOVL C01803 V=800.0 PL=0
MOVL C01804 V=800.0 PL=0
MOVL C01805 V=800.0 PL=0
MOVL C01806 V=800.0 PL=0
MOVL C01807 V=800.0 PL=0
MOVL C01808 V=800.0 PL=0
MOVL C01809 V=800.0 PL=0
MOVL C01810 V=800.0 PL=0
MOVL C01811 V=800.0 PL=0
MOVL C01812 V=800.0 PL=0
MOVL C01813 V=800.0 PL=0
MOVL C01814 V=800.0 PL=0
MOVL C01815 V=800.0 PL=0
MOVL C01816 V=800.0 PL=0
MOVL C01817 V=800.0 PL=0
MOVL C01818 V=800.0 PL=0
MOVL C01819 V=800.0 PL=0
MOVL C01820 V=800.0 PL=0
MOVL C01821 V=800.0 PL=0
MOVL C01822 V=800.0 PL=0
MOVL C01823 V=800.0 PL=0
MOVL C01824 V=800.0 PL=0
MOVL C01825 V=800.0 PL=0
MOVL C01826 V=800.0 PL=0
MOVL C01827 V=800.0 PL=0
MOVL C01828 V=800.0 PL=0
MOVL C01829 V=800.0 PL=0
MOVL C01830 V=800.0 PL=0
MOVL C01831 V=800.0 PL=0
MOVL C01832 V=800.0 PL=0
MOVL C01833 V=800.0 PL=0
MOVL C01834 V=800.0 PL=0
MOVL C01835 V=800.0 PL=0
MOVL C01836 V=800.0 PL=0
MOVL C01837 V=800.0 PL=0
MOVL C01838 V=800.0 PL=0
MOVL C01839 V=800.0 PL=0
MOVL C01840 V=800.0 PL=0
MOVL C01841 V=800.0 PL=0
MOVL C01842 V=800.0 PL=0
MOVL C01843 V=800.0 PL=0
MOVL C01844 V=800.0 PL=0
MOVL C01845 V=800.0 PL=0
MOVL C01846 V=800.0 PL=0
MOVL C01847 V=800.0 PL=0
MOVL C01848 V=800.0 PL=0
MOVL C01849 V=800.0 PL=0
MOVL C01850 V=800.0 PL=0
MOVL C01851 V=800.0 PL=0
MOVL C01852 V=800.0 PL=0
MOVL C01853 V=800.0 PL=0
MOVL C01854 V=800.0 PL=0
MOVL C01855 V=800.0 PL=0
MOVL C01856 V=800.0 PL=0
MOVL C01857 V=800.0 PL=0
MOVL C01858 V=800.0 PL=0
MOVL C01859 V=800.0 PL=0
MOVL C01860 V=800.0 PL=0
MOVL C01861 V=800.0 PL=0
MOVL C01862 V=800.0 PL=0
MOVL C01863 V=800.0 PL=0
MOVL C01864 V=800.0 PL=0
MOVL C01865 V=800.0 PL=0
MOVL C01866 V=800.0 PL=0
MOVL C01867 V=800.0 PL=0
MOVL C01868 V=800.0 PL=0
MOVL C01869 V=800.0 PL=0
MOVL C01870 V=800.0 PL=0
MOVL C01871 V=800.0 PL=0
MOVL C01872 V=800.0 PL=0
MOVL C01873 V=800.0 PL=0
MOVL C01874 V=800.0 PL=0
MOVL C01875 V=800.0 PL=0
MOVL C01876 V=800.0 PL=0
MOVL C01877 V=800.0 PL=0
MOVL C01878 V=800.0 PL=0
MOVL C01879 V=800.0 PL=0
MOVL C01880 V=800.0 PL=0
MOVL C01881 V=800.0 PL=0
MOVL C01882 V=800.0 PL=0
MOVL C01883 V=800.0 PL=0
MOVL C01884 V=800.0 PL=0
MOVL C01885 V=800.0 PL=0
MOVL C01886 V=800.0 PL=0
MOVL C01887 V=800.0 PL=0
MOVL C01888 V=800.0 PL=0
MOVL C01889 V=800.0 PL=0
MOVL C01890 V=800.0 PL=0
MOVL C01891 V=800.0 PL=0
MOVL C01892 V=800.0 PL=0
MOVL C01893 V=800.0 PL=0
MOVL C01894 V=800.0 PL=0
MOVL C01895 V=800.0 PL=0
MOVL C01896 V=800.0 PL=0
MOVL C01897 V=800.0 PL=0
MOVL C01898 V=800.0 PL=0
MOVL C01899 V=800.0 PL=0
MOVL C01900 V=800.0 PL=0
MOVL C01901 V=800.0 PL=0
MOVL C01902 V=800.0 PL=0
MOVL C01903 V=800.0 PL=0
MOVL C01904 V=800.0 PL=0
MOVL C01905 V=800.0 PL=0
MOVL C01906 V=800.0 PL=0
MOVL C01907 V=800.0 PL=0
MOVL C01908 V=800.0 PL=0
MOVL C01909 V=800.0 PL=0
MOVL C01910 V=800.0 PL=0
MOVL C01911 V=800.0 PL=0
MOVL C01912 V=800.0 PL=0
MOVL C01913 V=800.0 PL=0
MOVL C01914 V=800.0 PL=0
MOVL C01915 V=800.0 PL=0
MOVL C01916 V=800.0 PL=0
MOVL C01917 V=800.0 PL=0
MOVL C01918 V=800.0 PL=0
MOVL C01919 V=800.0 PL=0
MOVL C01920 V=800.0 PL=0
MOVL C01921 V=800.0 PL=0
MOVL C01922 V=800.0 PL=0
MOVL C01923 V=800.0 PL=0
MOVL C01924 V=800.0 PL=0
MOVL C01925 V=800.0 PL=0
MOVL C01926 V=800.0 PL=0
MOVL C01927 V=800.0 PL=0
MOVL C01928 V=800.0 PL=0
MOVL C01929 V=800.0 PL=0
MOVL C01930 V=800.0 PL=0
MOVL C01931 V=800.0 PL=0
MOVL C01932 V=800.0 PL=0
MOVL C01933 V=800.0 PL=0
MOVL C01934 V=800.0 PL=0
MOVL C01935 V=800.0 PL=0
MOVL C01936 V=800.0 PL=0
MOVL C01937 V=800.0 PL=0
MOVL C01938 V=800.0 PL=0
MOVL C01939 V=800.0 PL=0
MOVL C01940 V=800.0 PL=0
MOVL C01941 V=800.0 PL=0
MOVL C01942 V=800.0 PL=0
MOVL C01943 V=800.0 PL=0
MOVL C01944 V=800.0 PL=0
MOVL C01945 V=800.0 PL=0
MOVL C01946 V=800.0 PL=0
MOVL C01947 V=800.0 PL=0
MOVL C01948 V=800.0 PL=0
MOVL C01949 V=800.0 PL=0
MOVL C01950 V=800.0 PL=0
MOVL C01951 V=800.0 PL=0
MOVL C01952 V=800.0 PL=0
MOVL C01953 V=800.0 PL=0
MOVL C01954 V=800.0 PL=0
MOVL C01955 V=800.0 PL=0
MOVL C01956 V=800.0 PL=0
MOVL C01957 V=800.0 PL=0
MOVL C01958 V=800.0 PL=0
MOVL C01959 V=800.0 PL=0
MOVL C01960 V=800.0 PL=0
MOVL C01961 V=800.0 PL=0
MOVL C01962 V=800.0 PL=0
MOVL C01963 V=800.0 PL=0
MOVL C01964 V=800.0 PL=0
MOVL C01965 V=800.0 PL=0
MOVL C01966 V=800.0 PL=0
MOVL C01967 V=800.0 PL=0
MOVL C01968 V=800.0 PL=0
MOVL C01969 V=800.0 PL=0
MOVL C01970 V=800.0 PL=0
MOVL C01971 V=800.0 PL=0
MOVL C01972 V=800.0 PL=0
MOVL C01973 V=800.0 PL=0
MOVL C01974 V=800.0 PL=0
MOVL C01975 V=800.0 PL=0
MOVL C01976 V=800.0 PL=0
MOVL C01977 V=800.0 PL=0
MOVL C01978 V=800.0 PL=0
MOVL C01979 V=800.0 PL=0
MOVL C01980 V=800.0 PL=0
MOVL C01981 V=800.0 PL=0
MOVL C01982 V=800.0 PL=0
MOVL C01983 V=800.0 PL=0
MOVL C01984 V=800.0 PL=0
MOVL C01985 V=800.0 PL=0
MOVL C01986 V=800.0 PL=0
MOVL C01987 V=800.0 PL=0
MOVL C01988 V=800.0 PL=0
MOVL C01989 V=800.0 PL=0
MOVL C01990 V=800.0 PL=0
MOVL C01991 V=800.0 PL=0
MOVL C01992 V=800.0 PL=0
MOVL C01993 V=800.0 PL=0
MOVL C01994 V=800.0 PL=0
MOVL C01995 V=800.0 PL=0
MOVL C01996 V=800.0 PL=0
MOVL C01997 V=800.0 PL=0
MOVL C01998 V=800.0 PL=0
MOVL C01999 V=800.0 PL=0
MOVL C02000 V=800.0 PL=0
MOVL C02001 V=800.0 PL=0
MOVL C02002 V=800.0 PL=0
MOVL C02003 V=800.0 PL=0
MOVL C02004 V=800.0 PL=0
MOVL C02005 V=800.0 PL=0
MOVL C02006 V=800.0 PL=0
MOVL C02007 V=800.0 PL=0
MOVL C02008 V=800.0 PL=0
MOVL C02009 V=800.0 PL=0
MOVL C02010 V=800.0 PL=0
MOVL C02011 V=800.0 PL=0
MOVL C02012 V=800.0 PL=0
MOVL C02013 V=800.0 PL=0
MOVL C02014 V=800.0 PL=0
MOVL C02015 V=800.0 PL=0
MOVL C02016 V=800.0 PL=0
MOVL C02017 V=800.0 PL=0
MOVL C02018 V=800.0 PL=0
MOVL C02019 V=800.0 PL=0
MOVL C02020 V=800.0 PL=0
MOVL C02021 V=800.0 PL=0
MOVL C02022 V=800.0 PL=0
MOVL C02023 V=800.0 PL=0
MOVL C02024 V=800.0 PL=0
MOVL C02025 V=800.0 PL=0
MOVL C02026 V=800.0 PL=0
MOVL C02027 V=800.0 PL=0
MOVL C02028 V=800.0 PL=0
MOVL C02029 V=800.0 PL=0
MOVL C02030 V=800.0 PL=0
MOVL C02031 V=800.0 PL=0
MOVL C02032 V=800.0 PL=0
MOVL C02033 V=800.0 PL=0
MOVL C02034 V=800.0 PL=0
MOVL C02035 V=800.0 PL=0
MOVL C02036 V=800.0 PL=0
MOVL C02037 V=800.0 PL=0
MOVL C02038 V=800.0 PL=0
MOVL C02039 V=800.0 PL=0
